// TIA Portal project "HydroPlantProject" (V15)

(* hardware
DEVICE "S71500/ET200MP station_1"  S7-1500 station
   slot 0: "Rail_0"  Rack  6ES7 590-1***0-0AA0
   slot 1: "PLC_1"  CPU 1511-1 PN  6ES7 511-1AK00-0AB0  V1.8
      slot 3: "CPU display_1"  6ES7591-1AA00-0AA0
DEVICE "PC-System_1"  SIMATIC PC station
   slot 0: "SIMATIC PC station"  Rail  SIMATIC PC-Station  V1.0
      slot 125: "Stationmanager"  Station_Manager  V6.0.4
   slot 1: "HMI_RT_1"  WinCC RT Professional  6AV2 105-0xxxx-xxxx  15.0.0.0
   slot 2: "IE general_1"  IE General  IE_CP  V8.2.0
*)

// ===== PLC "PLC_1"  CPU 1511-1 PN =====

VAR_GLOBAL   // PLC tag table "Default tag table"
   "Brake_Out" AT %M4.0 : Bool;
   "OilPumpVFDsp_Out" AT %MW6 : Int;
   "OilTemp_In" AT %MW12 : Int;
   "kW_In" AT %MW14 : Int;
   "RPM_In" AT %MW16 : Int;
   "Baffle_Out" AT %MW18 : Int;
   "OilPumpVFDen_Out" AT %M4.1 : Bool;
   "ProgLang" AT %MW0 : Int;
   "ONS1" AT %M2.0 : Bool;
   "PB_LAD" AT %M2.1 : Bool;
   "ONS" AT %M2.2 : Bool;
   "ONS2" AT %M2.3 : Bool;
   "ONS3" AT %M2.4 : Bool;
   "PB_FBD" AT %M2.5 : Bool;
   "PB_SCL" AT %M2.6 : Bool;
   "PB_STL" AT %M2.7 : Bool;
   "AlarmHorn_Out" AT %M3.0 : Bool;
   "StationInterlock_Out" AT %M3.1 : Bool;
   "OilPumpVFDpct" AT %MW8 : Int;
   "BafflePct" AT %MW10 : Int;
   "OilTemp" AT %MW20 : Int;
   "OilFlow" AT %MW22 : Int;
   "OilFlow_In" AT %MW24 : Int;
   "RPM" AT %MW26 : Int;
   "Current" AT %MW28 : Int;
   "Current_In" AT %MW30 : Int;
   "OilPumpVFDoff_Pb" AT %M3.2 : Bool;
   "OilPumpVFDhand_Pb" AT %M3.3 : Bool;
   "OilPumpVFDauto_Pb" AT %M3.4 : Bool;
   "BrakeOff_Pb" AT %M3.5 : Bool;
   "BrakeHand_Pb" AT %M3.6 : Bool;
   "BrakeAuto_Pb" AT %M3.7 : Bool;
   "BrakeHoa" AT %MW34 : Int;
   "AlarmHornOff_Pb" AT %M4.2 : Bool;
   "AlarmHornHand_Pb" AT %M4.3 : Bool;
   "AlarmHornAuto_Pb" AT %M4.4 : Bool;
   "AlarmHornHoa" AT %MW36 : Int;
   "StationIntOff_Pb" AT %M4.5 : Bool;
   "StationIntHand_Pb" AT %M4.6 : Bool;
   "StationIntAuto_Pb" AT %M4.7 : Bool;
   "StationIntHoa" AT %MW38 : Int;
   "OilPumpVFD_Ctrl" AT %M5.0 : Bool;
   "StationIntl_Ctrl" AT %M5.1 : Bool;
   "AlarmHorn_Ctrl" AT %M5.2 : Bool;
   "Brake_Ctrl" AT %M5.3 : Bool;
   "OilLowFlowDelay_Sp" AT %MW40 : Int;
   "AlarmReset" AT %M5.4 : Bool;
   "AlarmSilence" AT %M5.5 : Bool;
   "OilLowFlowAlarm" AT %M5.6 : Bool;
   "OilLowFlowNotify" AT %M5.7 : Bool;
   "OilLLflowSp" AT %MW42 : Int;
   "OvercurrentDelay_Sp" AT %MW44 : Int;
   "OvercurrentSp" AT %MW46 : Int;
   "OvercurrentAlarm" AT %M48.0 : Bool;
   "OvercurrentNotify" AT %M48.1 : Bool;
   "HighOilTempDelay_Sp" AT %MW50 : Int;
   "HighOilTempAlarm" AT %M48.2 : Bool;
   "HighOilTempNotify" AT %M48.3 : Bool;
   "HighOilTempSp" AT %MW52 : Int;
   "OverspeedDelay_Sp" AT %MW54 : Int;
   "OverspeedSp" AT %MW56 : Int;
   "OverspeedAlarm" AT %M48.4 : Bool;
   "OverspeedNotify" AT %M48.5 : Bool;
   "OilHighFlowDelay_Sp" AT %MW58 : Int;
   "OilHHflowSp" AT %MW60 : Int;
   "OilHighFlowAlarm" AT %M48.6 : Bool;
   "OilHighFlowNotify" AT %M48.7 : Bool;
   "BrakeFailureDelay_Sp" AT %MW62 : Int;
   "BrakeFailureAlarm" AT %M49.0 : Bool;
   "BrakeFailureNotify" AT %M49.1 : Bool;
   "EStop" AT %M49.2 : Bool;
   "EStopAlarm" AT %M49.3 : Bool;
   "EStopNotify" AT %M49.4 : Bool;
   "Tag_1" AT %T1 : Timer;
   "Tag_2" AT %T2 : Timer;
   "ONS2(1)" AT %M49.5 : Bool;
   "ONS2(2)" AT %M49.6 : Bool;
   "Baffle_En" AT %M49.7 : Bool;
   "Deleteme" AT %M64.0 : Bool;
   "deleteme1" AT %MD66 : Real;
   "WarmupMode" AT %M64.1 : Bool;
   "StabilizeMode" AT %M64.2 : Bool;
   "GenerationMode" AT %M64.3 : Bool;
   "CooldownMode" AT %M64.4 : Bool;
   "IdleMode" AT %M64.5 : Bool;
   "FaultMode" AT %M64.6 : Bool;
   "WarmupRPM" AT %MW70 : Int;
   "BafflePIDSp" AT %MW72 : Int;
   "BaffleHOA" AT %MW74 : Int;
   "Baffle_Ctrl" AT %M64.7 : Bool;
   "VFD_Sp" AT %MW76 : Int;
   "WarmupVFDpct" AT %MW78 : Int;
   "WarmupOilTemp" AT %MW80 : Int;
   "WarmupOilTempDelaySp" AT %MW82 : Int;
   "WarmupTrasition" AT %M65.0 : Bool;
   "BafflePIDin" AT %MW84 : Int;
   "StabilizekWSp" AT %MW86 : Int;
   "StabilizeDelaySp" AT %MW88 : Int;
   "StabilizeTrasition" AT %M65.1 : Bool;
   "SystemStart_Pb" AT %M65.2 : Bool;
   "StartSequenceBit" AT %M65.3 : Bool;
   "SystemStop_Pb" AT %M65.4 : Bool;
   "GenerationTransition" AT %M65.5 : Bool;
   "CooldownRPM" AT %MW90 : Int;
   "CooldownDelaySp" AT %MW92 : Int;
   "CooldownTrasition" AT %M65.6 : Bool;
   "CooldownRPMSp" AT %MW94 : Int;
   "CooldownOilTempSp" AT %MW96 : Int;
   "ONS4" AT %M65.7 : Bool;
   "SequenceRunning" AT %M98.0 : Bool;
   "ONS5" AT %M98.1 : Bool;
   "HOFoverrideVFDsp" AT %MW100 : Int;
   "ONS6" AT %M98.2 : Bool;
   "BaffleManual" AT %M98.3 : Bool;
   "BaffleAuto_Pb" AT %M98.4 : Bool;
   "BaffleHand_Pb" AT %M98.5 : Bool;
   "BaffleOff_Pb" AT %M98.6 : Bool;
   "ONS8" AT %M98.7 : Bool;
   "BaffleManualSp" AT %MD102 : Real;
   "ONS9" AT %M99.0 : Bool;
   "ONS10" AT %M99.1 : Bool;
   "ONS7" AT %M99.2 : Bool;
   "VFDHand_Pb" AT %M99.3 : Bool;
   "VFDOff_Pb" AT %M99.4 : Bool;
   "VFDAuto_Pb" AT %M99.5 : Bool;
   "ONS11" AT %M99.6 : Bool;
   "ONS12" AT %M99.7 : Bool;
   "ONS13" AT %M106.0 : Bool;
   "VFDHOA" AT %MW108 : Int;
   "VFDManualSp" AT %MD110 : Real;
   "ONS14" AT %M106.1 : Bool;
   "ONS15" AT %M106.2 : Bool;
   "VFDmanual" AT %M106.3 : Bool;
   "OilPumpVFDon" AT %M106.4 : Bool;
   "BafflePID_On" AT %M106.5 : Bool;
   "FullAutoBit" AT %M106.6 : Bool;
   "HM_Minutes" AT %MW32 : Int;
   "HM_Hours" AT %MW114 : Int;
   "HM_Days" AT %MW116 : Int;
   "ResetHourmeter_Pb" AT %M106.7 : Bool;
   "ModeInt" AT %MW118 : Int;
END_VAR

DATA_BLOCK "SimLogic_DB"   // DB1
{ S7_Optimized_Access := 'TRUE' }
VERSION : 0.1
// stored: InstanceOfName SimLogic
"SimLogic"
BEGIN
END_DATA_BLOCK

DATA_BLOCK "MODES_LAD_DB"   // DB2
{ S7_Optimized_Access := 'TRUE' }
VERSION : 0.1
// stored: InstanceOfName MODES_LAD
"MODES_LAD"
BEGIN
END_DATA_BLOCK

DATA_BLOCK "MODES_FBD_DB"   // DB4
{ S7_Optimized_Access := 'TRUE' }
VERSION : 0.1
// stored: InstanceOfName MODES_FBD
"MODES_FBD"
BEGIN
END_DATA_BLOCK

DATA_BLOCK "IO_LAD_DB"   // DB5
{ S7_Optimized_Access := 'TRUE' }
VERSION : 0.1
// stored: InstanceOfName IO_LAD
"IO_LAD"
BEGIN
END_DATA_BLOCK

DATA_BLOCK "IO_FBD_DB"   // DB6
{ S7_Optimized_Access := 'TRUE' }
VERSION : 0.1
// stored: InstanceOfName IO_FBD
"IO_FBD"
BEGIN
END_DATA_BLOCK

DATA_BLOCK "IO_SCL_DB"   // DB7
{ S7_Optimized_Access := 'TRUE' }
VERSION : 0.1
// stored: InstanceOfName IO_SCL
"IO_SCL"
BEGIN
END_DATA_BLOCK

DATA_BLOCK "IO_STL_DB"   // DB8
{ S7_Optimized_Access := 'TRUE' }
VERSION : 0.1
// stored: InstanceOfName IO_STL
"IO_STL"
BEGIN
END_DATA_BLOCK

DATA_BLOCK "ALARMS_LAD_DB"   // DB9
{ S7_Optimized_Access := 'TRUE' }
VERSION : 0.1
// stored: InstanceOfName ALARMS_LAD
"ALARMS_LAD"
BEGIN
END_DATA_BLOCK

DATA_BLOCK "HOA_LAD_DB"   // DB10
{ S7_Optimized_Access := 'TRUE' }
VERSION : 0.1
// stored: InstanceOfName HOA_LAD
"HOA_LAD"
BEGIN
END_DATA_BLOCK

DATA_BLOCK "HOA_FBD_DB"   // DB11
{ S7_Optimized_Access := 'TRUE' }
VERSION : 0.1
// stored: InstanceOfName HOA_FBD
"HOA_FBD"
BEGIN
END_DATA_BLOCK

DATA_BLOCK "HOA_SCL_DB"   // DB12
{ S7_Optimized_Access := 'TRUE' }
VERSION : 0.1
// stored: InstanceOfName HOA_SCL
"HOA_SCL"
BEGIN
END_DATA_BLOCK

DATA_BLOCK "HOA_STL_DB"   // DB13
{ S7_Optimized_Access := 'TRUE' }
VERSION : 0.1
// stored: InstanceOfName HOA_STL
"HOA_STL"
BEGIN
END_DATA_BLOCK

DATA_BLOCK "ALARMS_FBD_DB"   // DB14
{ S7_Optimized_Access := 'TRUE' }
VERSION : 0.1
// stored: InstanceOfName ALARMS_FBD
"ALARMS_FBD"
BEGIN
END_DATA_BLOCK

DATA_BLOCK "ALARMS_SCL_DB"   // DB15
{ S7_Optimized_Access := 'TRUE' }
VERSION : 0.1
// stored: InstanceOfName ALARMS_SCL
"ALARMS_SCL"
BEGIN
END_DATA_BLOCK

DATA_BLOCK "ALARMS_STL_DB"   // DB16
{ S7_Optimized_Access := 'TRUE' }
VERSION : 0.1
// stored: InstanceOfName ALARMS_STL
"ALARMS_STL"
BEGIN
END_DATA_BLOCK

DATA_BLOCK "MODES_SCL_DB"   // DB44
{ S7_Optimized_Access := 'TRUE' }
VERSION : 0.1
// stored: InstanceOfName MODES_SCL
"MODES_SCL"
BEGIN
END_DATA_BLOCK

DATA_BLOCK "MODES_STL_DB"   // DB45
{ S7_Optimized_Access := 'TRUE' }
VERSION : 0.1
// stored: InstanceOfName MODES_STL
"MODES_STL"
BEGIN
END_DATA_BLOCK

DATA_BLOCK "SEQUENCE_DB"   // DB58
{ S7_Optimized_Access := 'TRUE' }
VERSION : 0.1
// stored: InstanceOfName SEQUENCE
"SEQUENCE"
BEGIN
END_DATA_BLOCK

DATA_BLOCK "HOURMETER_LAD_DB"   // DB61
{ S7_Optimized_Access := 'TRUE' }
VERSION : 0.1
// stored: InstanceOfName HOURMETER_LAD
"HOURMETER_LAD"
BEGIN
END_DATA_BLOCK

DATA_BLOCK "HOURMETER_FBD_DB"   // DB62
{ S7_Optimized_Access := 'TRUE' }
VERSION : 0.1
// stored: InstanceOfName HOURMETER_FBD
"HOURMETER_FBD"
BEGIN
END_DATA_BLOCK

DATA_BLOCK "HOURMETER_SCL_DB"   // DB63
{ S7_Optimized_Access := 'TRUE' }
VERSION : 0.1
// stored: InstanceOfName HOURMETER_SCL
"HOURMETER_SCL"
BEGIN
END_DATA_BLOCK

DATA_BLOCK "HOURMETER_STL_DB"   // DB64
{ S7_Optimized_Access := 'TRUE' }
VERSION : 0.1
// stored: InstanceOfName HOURMETER_STL
"HOURMETER_STL"
BEGIN
END_DATA_BLOCK

// folder: System blocks/Program resources

DATA_BLOCK "IEC_Timer_0_DB_25"   // DB3
{ S7_Optimized_Access := 'TRUE' }
AUTHOR : Simatic
FAMILY : IEC
NAME : IEC_TMR
VERSION : 1.0
// stored: InstanceOfName IEC_TIMER
"IEC_TIMER"
BEGIN
END_DATA_BLOCK

DATA_BLOCK "IEC_Timer_0_DB"   // DB17
{ S7_Optimized_Access := 'TRUE' }
AUTHOR : Simatic
FAMILY : IEC
NAME : IEC_TMR
VERSION : 1.0
// stored: InstanceOfName IEC_TIMER
"IEC_TIMER"
BEGIN
END_DATA_BLOCK

DATA_BLOCK "IEC_Timer_0_DB_1"   // DB18
{ S7_Optimized_Access := 'TRUE' }
AUTHOR : Simatic
FAMILY : IEC
NAME : IEC_TMR
VERSION : 1.0
// stored: InstanceOfName IEC_TIMER
"IEC_TIMER"
BEGIN
END_DATA_BLOCK

DATA_BLOCK "IEC_Timer_0_DB_2"   // DB19
{ S7_Optimized_Access := 'TRUE' }
AUTHOR : Simatic
FAMILY : IEC
NAME : IEC_TMR
VERSION : 1.0
// stored: InstanceOfName IEC_TIMER
"IEC_TIMER"
BEGIN
END_DATA_BLOCK

DATA_BLOCK "IEC_Timer_0_DB_3"   // DB20
{ S7_Optimized_Access := 'TRUE' }
AUTHOR : Simatic
FAMILY : IEC
NAME : IEC_TMR
VERSION : 1.0
// stored: InstanceOfName IEC_TIMER
"IEC_TIMER"
BEGIN
END_DATA_BLOCK

DATA_BLOCK "IEC_Timer_0_DB_4"   // DB21
{ S7_Optimized_Access := 'TRUE' }
AUTHOR : Simatic
FAMILY : IEC
NAME : IEC_TMR
VERSION : 1.0
// stored: InstanceOfName IEC_TIMER
"IEC_TIMER"
BEGIN
END_DATA_BLOCK

DATA_BLOCK "IEC_Timer_0_DB_5"   // DB22
{ S7_Optimized_Access := 'TRUE' }
AUTHOR : Simatic
FAMILY : IEC
NAME : IEC_TMR
VERSION : 1.0
// stored: InstanceOfName IEC_TIMER
"IEC_TIMER"
BEGIN
END_DATA_BLOCK

DATA_BLOCK "IEC_Timer_0_DB_6"   // DB23
{ S7_Optimized_Access := 'TRUE' }
AUTHOR : Simatic
FAMILY : IEC
NAME : IEC_TMR
VERSION : 1.0
// stored: InstanceOfName IEC_TIMER
"IEC_TIMER"
BEGIN
END_DATA_BLOCK

DATA_BLOCK "IEC_Timer_0_DB_7"   // DB24
{ S7_Optimized_Access := 'TRUE' }
AUTHOR : Simatic
FAMILY : IEC
NAME : IEC_TMR
VERSION : 1.0
// stored: InstanceOfName IEC_TIMER
"IEC_TIMER"
BEGIN
END_DATA_BLOCK

DATA_BLOCK "IEC_Timer_0_DB_8"   // DB25
{ S7_Optimized_Access := 'TRUE' }
AUTHOR : Simatic
FAMILY : IEC
NAME : IEC_TMR
VERSION : 1.0
// stored: InstanceOfName IEC_TIMER
"IEC_TIMER"
BEGIN
END_DATA_BLOCK

DATA_BLOCK "IEC_Timer_0_DB_9"   // DB26
{ S7_Optimized_Access := 'TRUE' }
AUTHOR : Simatic
FAMILY : IEC
NAME : IEC_TMR
VERSION : 1.0
// stored: InstanceOfName IEC_TIMER
"IEC_TIMER"
BEGIN
END_DATA_BLOCK

DATA_BLOCK "IEC_Timer_0_DB_10"   // DB27
{ S7_Optimized_Access := 'TRUE' }
AUTHOR : Simatic
FAMILY : IEC
NAME : IEC_TMR
VERSION : 1.0
// stored: InstanceOfName IEC_TIMER
"IEC_TIMER"
BEGIN
END_DATA_BLOCK

DATA_BLOCK "IEC_Timer_0_DB_110"   // DB28
{ S7_Optimized_Access := 'TRUE' }
AUTHOR : Simatic
FAMILY : IEC
NAME : IEC_TMR
VERSION : 1.0
// stored: InstanceOfName IEC_TIMER
"IEC_TIMER"
BEGIN
END_DATA_BLOCK

DATA_BLOCK "IEC_Timer_0_DB_11"   // DB29
{ S7_Optimized_Access := 'TRUE' }
AUTHOR : Simatic
FAMILY : IEC
NAME : IEC_TMR
VERSION : 1.0
// stored: InstanceOfName IEC_TIMER
"IEC_TIMER"
BEGIN
END_DATA_BLOCK

DATA_BLOCK "IEC_Timer_0_DB_12"   // DB30
{ S7_Optimized_Access := 'TRUE' }
AUTHOR : Simatic
FAMILY : IEC
NAME : IEC_TMR
VERSION : 1.0
// stored: InstanceOfName IEC_TIMER
"IEC_TIMER"
BEGIN
END_DATA_BLOCK

DATA_BLOCK "IEC_Timer_0_DB_13"   // DB31
{ S7_Optimized_Access := 'TRUE' }
AUTHOR : Simatic
FAMILY : IEC
NAME : IEC_TMR
VERSION : 1.0
// stored: InstanceOfName IEC_TIMER
"IEC_TIMER"
BEGIN
END_DATA_BLOCK

DATA_BLOCK "IEC_Timer_0_DB_14"   // DB32
{ S7_Optimized_Access := 'TRUE' }
AUTHOR : Simatic
FAMILY : IEC
NAME : IEC_TMR
VERSION : 1.0
// stored: InstanceOfName IEC_TIMER
"IEC_TIMER"
BEGIN
END_DATA_BLOCK

DATA_BLOCK "IEC_Timer_0_DB_15"   // DB33
{ S7_Optimized_Access := 'TRUE' }
AUTHOR : Simatic
FAMILY : IEC
NAME : IEC_TMR
VERSION : 1.0
// stored: InstanceOfName IEC_TIMER
"IEC_TIMER"
BEGIN
END_DATA_BLOCK

DATA_BLOCK "IEC_Timer_0_DB_16"   // DB34
{ S7_Optimized_Access := 'TRUE' }
AUTHOR : Simatic
FAMILY : IEC
NAME : IEC_TMR
VERSION : 1.0
// stored: InstanceOfName IEC_TIMER
"IEC_TIMER"
BEGIN
END_DATA_BLOCK

DATA_BLOCK "IEC_Timer_0_DB_17"   // DB35
{ S7_Optimized_Access := 'TRUE' }
AUTHOR : Simatic
FAMILY : IEC
NAME : IEC_TMR
VERSION : 1.0
// stored: InstanceOfName IEC_TIMER
"IEC_TIMER"
BEGIN
END_DATA_BLOCK

DATA_BLOCK "IEC_Timer_0_DB_18"   // DB36
{ S7_Optimized_Access := 'TRUE' }
AUTHOR : Simatic
FAMILY : IEC
NAME : IEC_TMR
VERSION : 1.0
// stored: InstanceOfName IEC_TIMER
"IEC_TIMER"
BEGIN
END_DATA_BLOCK

DATA_BLOCK "IEC_Timer_0_DB_19"   // DB37
{ S7_Optimized_Access := 'TRUE' }
AUTHOR : Simatic
FAMILY : IEC
NAME : IEC_TMR
VERSION : 1.0
// stored: InstanceOfName IEC_TIMER
"IEC_TIMER"
BEGIN
END_DATA_BLOCK

DATA_BLOCK "IEC_Timer_0_DB_20"   // DB38
{ S7_Optimized_Access := 'TRUE' }
AUTHOR : Simatic
FAMILY : IEC
NAME : IEC_TMR
VERSION : 1.0
// stored: InstanceOfName IEC_TIMER
"IEC_TIMER"
BEGIN
END_DATA_BLOCK

DATA_BLOCK "IEC_Timer_0_DB_21"   // DB39
{ S7_Optimized_Access := 'TRUE' }
AUTHOR : Simatic
FAMILY : IEC
NAME : IEC_TMR
VERSION : 1.0
// stored: InstanceOfName IEC_TIMER
"IEC_TIMER"
BEGIN
END_DATA_BLOCK

DATA_BLOCK "IEC_Timer_0_DB_22"   // DB40
{ S7_Optimized_Access := 'TRUE' }
AUTHOR : Simatic
FAMILY : IEC
NAME : IEC_TMR
VERSION : 1.0
// stored: InstanceOfName IEC_TIMER
"IEC_TIMER"
BEGIN
END_DATA_BLOCK

DATA_BLOCK "IEC_Timer_0_DB_23"   // DB41
{ S7_Optimized_Access := 'TRUE' }
AUTHOR : Simatic
FAMILY : IEC
NAME : IEC_TMR
VERSION : 1.0
// stored: InstanceOfName IEC_TIMER
"IEC_TIMER"
BEGIN
END_DATA_BLOCK

DATA_BLOCK "IEC_Timer_1_DB"   // DB43
{ S7_Optimized_Access := 'TRUE' }
AUTHOR : Simatic
FAMILY : IEC
NAME : IEC_TMR
VERSION : 1.0
// stored: InstanceOfName IEC_TIMER
"IEC_TIMER"
BEGIN
END_DATA_BLOCK

DATA_BLOCK "IEC_Timer_0_DB_24"   // DB46
{ S7_Optimized_Access := 'TRUE' }
AUTHOR : Simatic
FAMILY : IEC
NAME : IEC_TMR
VERSION : 1.0
// stored: InstanceOfName IEC_TIMER
"IEC_TIMER"
BEGIN
END_DATA_BLOCK

DATA_BLOCK "IEC_Timer_0_DB_26"   // DB47
{ S7_Optimized_Access := 'TRUE' }
AUTHOR : Simatic
FAMILY : IEC
NAME : IEC_TMR
VERSION : 1.0
// stored: InstanceOfName IEC_TIMER
"IEC_TIMER"
BEGIN
END_DATA_BLOCK

DATA_BLOCK "IEC_Timer_0_DB_27"   // DB48
{ S7_Optimized_Access := 'TRUE' }
AUTHOR : Simatic
FAMILY : IEC
NAME : IEC_TMR
VERSION : 1.0
// stored: InstanceOfName IEC_TIMER
"IEC_TIMER"
BEGIN
END_DATA_BLOCK

DATA_BLOCK "IEC_Timer_0_DB_28"   // DB49
{ S7_Optimized_Access := 'TRUE' }
AUTHOR : Simatic
FAMILY : IEC
NAME : IEC_TMR
VERSION : 1.0
// stored: InstanceOfName IEC_TIMER
"IEC_TIMER"
BEGIN
END_DATA_BLOCK

DATA_BLOCK "IEC_Timer_0_DB_29"   // DB50
{ S7_Optimized_Access := 'TRUE' }
AUTHOR : Simatic
FAMILY : IEC
NAME : IEC_TMR
VERSION : 1.0
// stored: InstanceOfName IEC_TIMER
"IEC_TIMER"
BEGIN
END_DATA_BLOCK

DATA_BLOCK "IEC_Timer_0_DB_30"   // DB51
{ S7_Optimized_Access := 'TRUE' }
AUTHOR : Simatic
FAMILY : IEC
NAME : IEC_TMR
VERSION : 1.0
// stored: InstanceOfName IEC_TIMER
"IEC_TIMER"
BEGIN
END_DATA_BLOCK

DATA_BLOCK "IEC_Timer_0_DB_31"   // DB52
{ S7_Optimized_Access := 'TRUE' }
AUTHOR : Simatic
FAMILY : IEC
NAME : IEC_TMR
VERSION : 1.0
// stored: InstanceOfName IEC_TIMER
"IEC_TIMER"
BEGIN
END_DATA_BLOCK

DATA_BLOCK "IEC_Timer_0_DB_32"   // DB53
{ S7_Optimized_Access := 'TRUE' }
AUTHOR : Simatic
FAMILY : IEC
NAME : IEC_TMR
VERSION : 1.0
// stored: InstanceOfName IEC_TIMER
"IEC_TIMER"
BEGIN
END_DATA_BLOCK

DATA_BLOCK "IEC_Timer_0_DB_33"   // DB54
{ S7_Optimized_Access := 'TRUE' }
AUTHOR : Simatic
FAMILY : IEC
NAME : IEC_TMR
VERSION : 1.0
// stored: InstanceOfName IEC_TIMER
"IEC_TIMER"
BEGIN
END_DATA_BLOCK

DATA_BLOCK "IEC_Timer_0_DB_34"   // DB55
{ S7_Optimized_Access := 'TRUE' }
AUTHOR : Simatic
FAMILY : IEC
NAME : IEC_TMR
VERSION : 1.0
// stored: InstanceOfName IEC_TIMER
"IEC_TIMER"
BEGIN
END_DATA_BLOCK

DATA_BLOCK "IEC_Timer_0_DB_35"   // DB56
{ S7_Optimized_Access := 'TRUE' }
AUTHOR : Simatic
FAMILY : IEC
NAME : IEC_TMR
VERSION : 1.0
// stored: InstanceOfName IEC_TIMER
"IEC_TIMER"
BEGIN
END_DATA_BLOCK

DATA_BLOCK "IEC_Timer_0_DB_36"   // DB57
{ S7_Optimized_Access := 'TRUE' }
AUTHOR : Simatic
FAMILY : IEC
NAME : IEC_TMR
VERSION : 1.0
// stored: InstanceOfName IEC_TIMER
"IEC_TIMER"
BEGIN
END_DATA_BLOCK

DATA_BLOCK "IEC_Timer_0_DB_37"   // DB65
{ S7_Optimized_Access := 'TRUE' }
AUTHOR : Simatic
FAMILY : IEC
NAME : IEC_TMR
VERSION : 1.0
// stored: InstanceOfName IEC_TIMER
"IEC_TIMER"
BEGIN
END_DATA_BLOCK

DATA_BLOCK "IEC_Counter_0_DB"   // DB66
{ S7_Optimized_Access := 'TRUE' }
AUTHOR : Simatic
FAMILY : IEC
NAME : CNTR
VERSION : 1.0
// stored: InstanceOfName IEC_COUNTER
"IEC_COUNTER"
BEGIN
END_DATA_BLOCK

DATA_BLOCK "IEC_Counter_0_DB_1"   // DB67
{ S7_Optimized_Access := 'TRUE' }
AUTHOR : Simatic
FAMILY : IEC
NAME : CNTR
VERSION : 1.0
// stored: InstanceOfName IEC_COUNTER
"IEC_COUNTER"
BEGIN
END_DATA_BLOCK

DATA_BLOCK "IEC_Counter_0_DB_2"   // DB68
{ S7_Optimized_Access := 'TRUE' }
AUTHOR : Simatic
FAMILY : IEC
NAME : CNTR
VERSION : 1.0
// stored: InstanceOfName IEC_COUNTER
"IEC_COUNTER"
BEGIN
END_DATA_BLOCK

DATA_BLOCK "IEC_Timer_0_DB_38"   // DB69
{ S7_Optimized_Access := 'TRUE' }
AUTHOR : Simatic
FAMILY : IEC
NAME : IEC_TMR
VERSION : 1.0
// stored: InstanceOfName IEC_TIMER
"IEC_TIMER"
BEGIN
END_DATA_BLOCK

DATA_BLOCK "IEC_Timer_0_DB_39"   // DB70
{ S7_Optimized_Access := 'TRUE' }
AUTHOR : Simatic
FAMILY : IEC
NAME : IEC_TMR
VERSION : 1.0
// stored: InstanceOfName IEC_TIMER
"IEC_TIMER"
BEGIN
END_DATA_BLOCK

DATA_BLOCK "IEC_Timer_0_DB_40"   // DB71
{ S7_Optimized_Access := 'TRUE' }
AUTHOR : Simatic
FAMILY : IEC
NAME : IEC_TMR
VERSION : 1.0
// stored: InstanceOfName IEC_TIMER
"IEC_TIMER"
BEGIN
END_DATA_BLOCK

DATA_BLOCK "IEC_Counter_0_DB_3"   // DB72
{ S7_Optimized_Access := 'TRUE' }
AUTHOR : Simatic
FAMILY : IEC
NAME : CNTR
VERSION : 1.0
// stored: InstanceOfName IEC_COUNTER
"IEC_COUNTER"
BEGIN
END_DATA_BLOCK

DATA_BLOCK "IEC_Counter_0_DB_4"   // DB73
{ S7_Optimized_Access := 'TRUE' }
AUTHOR : Simatic
FAMILY : IEC
NAME : CNTR
VERSION : 1.0
// stored: InstanceOfName IEC_COUNTER
"IEC_COUNTER"
BEGIN
END_DATA_BLOCK

DATA_BLOCK "IEC_Counter_0_DB_5"   // DB74
{ S7_Optimized_Access := 'TRUE' }
AUTHOR : Simatic
FAMILY : IEC
NAME : CNTR
VERSION : 1.0
// stored: InstanceOfName IEC_COUNTER
"IEC_COUNTER"
BEGIN
END_DATA_BLOCK

DATA_BLOCK "IEC_Timer_0_DB_41"   // DB75
{ S7_Optimized_Access := 'TRUE' }
AUTHOR : Simatic
FAMILY : IEC
NAME : IEC_TMR
VERSION : 1.0
// stored: InstanceOfName IEC_TIMER
"IEC_TIMER"
BEGIN
END_DATA_BLOCK

DATA_BLOCK "IEC_Counter_0_DB_6"   // DB76
{ S7_Optimized_Access := 'TRUE' }
AUTHOR : Simatic
FAMILY : IEC
NAME : CNTR
VERSION : 1.0
// stored: InstanceOfName IEC_COUNTER
"IEC_COUNTER"
BEGIN
END_DATA_BLOCK

DATA_BLOCK "IEC_Counter_0_DB_7"   // DB77
{ S7_Optimized_Access := 'TRUE' }
AUTHOR : Simatic
FAMILY : IEC
NAME : CNTR
VERSION : 1.0
// stored: InstanceOfName IEC_COUNTER
"IEC_COUNTER"
BEGIN
END_DATA_BLOCK

DATA_BLOCK "IEC_Counter_0_DB_9"   // DB79
{ S7_Optimized_Access := 'TRUE' }
AUTHOR : Simatic
FAMILY : IEC
NAME : CNTR
VERSION : 1.0
// stored: InstanceOfName IEC_COUNTER
"IEC_COUNTER"
BEGIN
END_DATA_BLOCK

DATA_BLOCK "IEC_Timer_0_DB_42"   // DB80
{ S7_Optimized_Access := 'TRUE' }
AUTHOR : Simatic
FAMILY : IEC
NAME : IEC_TMR
VERSION : 1.0
// stored: InstanceOfName IEC_TIMER
"IEC_TIMER"
BEGIN
END_DATA_BLOCK

DATA_BLOCK "IEC_Timer_0_DB_43"   // DB81
{ S7_Optimized_Access := 'TRUE' }
AUTHOR : Simatic
FAMILY : IEC
NAME : IEC_TMR
VERSION : 1.0
// stored: InstanceOfName IEC_TIMER
"IEC_TIMER"
BEGIN
END_DATA_BLOCK

DATA_BLOCK "IEC_Counter_0_DB_10"   // DB82
{ S7_Optimized_Access := 'TRUE' }
AUTHOR : Simatic
FAMILY : IEC
NAME : CNTR
VERSION : 1.0
// stored: InstanceOfName IEC_COUNTER
"IEC_COUNTER"
BEGIN
END_DATA_BLOCK

DATA_BLOCK "IEC_Counter_0_DB_11"   // DB83
{ S7_Optimized_Access := 'TRUE' }
AUTHOR : Simatic
FAMILY : IEC
NAME : CNTR
VERSION : 1.0
// stored: InstanceOfName IEC_COUNTER
"IEC_COUNTER"
BEGIN
END_DATA_BLOCK

DATA_BLOCK "IEC_Counter_0_DB_12"   // DB84
{ S7_Optimized_Access := 'TRUE' }
AUTHOR : Simatic
FAMILY : IEC
NAME : CNTR
VERSION : 1.0
// stored: InstanceOfName IEC_COUNTER
"IEC_COUNTER"
BEGIN
END_DATA_BLOCK

DATA_BLOCK "IEC_Timer_0_DB_44"   // DB85
{ S7_Optimized_Access := 'TRUE' }
AUTHOR : Simatic
FAMILY : IEC
NAME : IEC_TMR
VERSION : 1.0
// stored: InstanceOfName IEC_TIMER
"IEC_TIMER"
BEGIN
END_DATA_BLOCK

// folder: (top level)

FUNCTION_BLOCK "SimLogic"   // FB1, LAD
{ S7_Optimized_Access := 'TRUE' }
VERSION : 0.1
   VAR
      "TO" : Bool;
      rpmv : Int;
      addrpmv : Bool;
      otsp : Int;
      ott : Int;
      TO1 : Bool;
      TO2 : Bool;
      be2 : Int;
      be3 : Int;
      be1 : Int;
      TO3 : Bool;
   END_VAR
   VAR_TEMP
      bf : Int;
      rpmvt : Int;
      bfr : Real;
   END_VAR
BEGIN

REGION Network 1
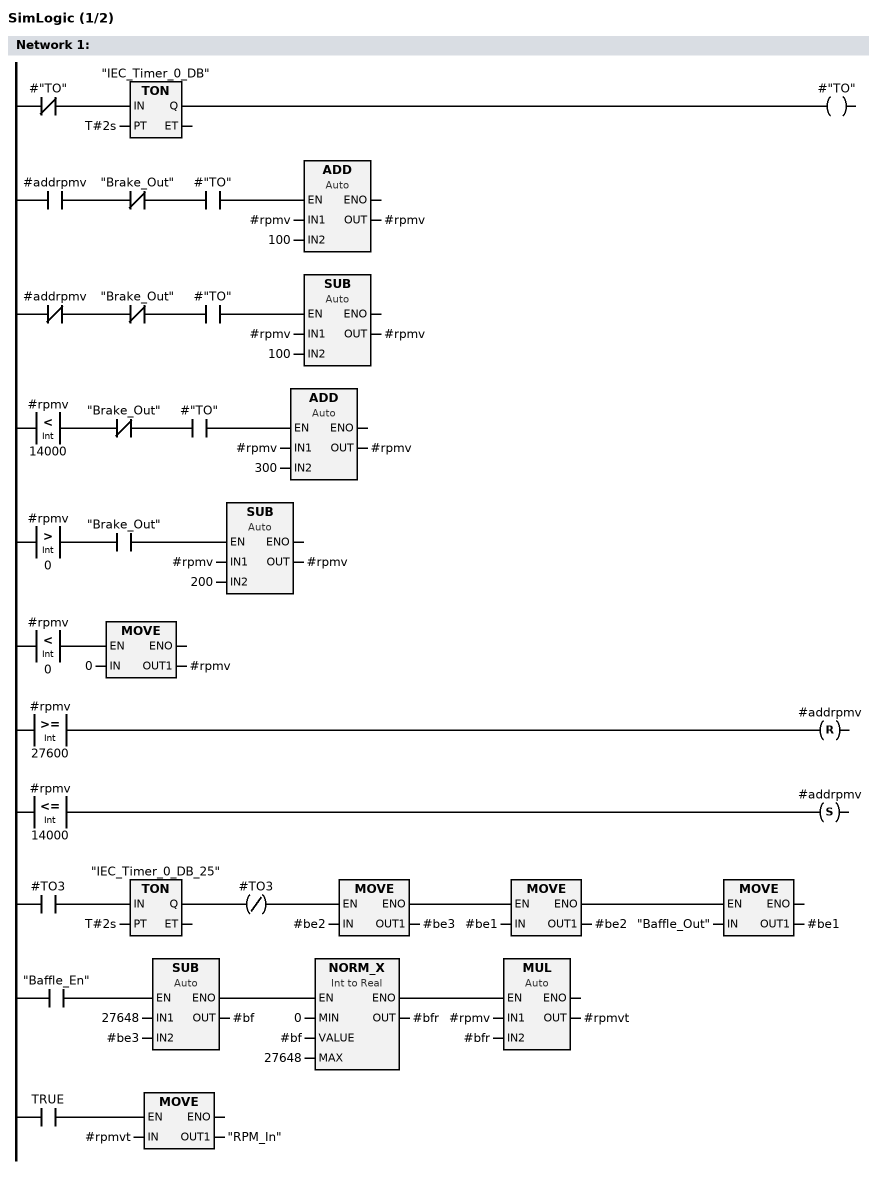
   "IEC_Timer_0_DB".TON(IN := NOT #"TO", PT := T#2s);
   #"TO" := "IEC_Timer_0_DB".Q;
   IF #addrpmv AND NOT "Brake_Out" AND #"TO" THEN #rpmv := #rpmv + 100; END_IF;
   IF NOT #addrpmv AND NOT "Brake_Out" AND #"TO" THEN #rpmv := #rpmv - 100; END_IF;
   IF (#rpmv < 14000) AND NOT "Brake_Out" AND #"TO" THEN #rpmv := #rpmv + 300; END_IF;
   IF (#rpmv > 0) AND "Brake_Out" THEN #rpmv := #rpmv - 200; END_IF;
   IF #rpmv < 0 THEN #rpmv := 0; END_IF;
   IF #rpmv >= 27600 THEN #addrpmv := FALSE; END_IF;
   IF #rpmv <= 14000 THEN #addrpmv := TRUE; END_IF;
   "IEC_Timer_0_DB_25".TON(IN := #TO3, PT := T#2s);
   #TO3 := NOT "IEC_Timer_0_DB_25".Q;
   IF "IEC_Timer_0_DB_25".Q THEN
       #be3 := #be2;
       #be2 := #be1;
       #be1 := "Baffle_Out";
   END_IF;
   IF "Baffle_En" THEN
       #bf := 27648 - #be3;
       #bfr := NORM_X(MIN := 0, VALUE := #bf, MAX := 27648);
       #rpmvt := #rpmv * #bfr;
   END_IF;
   IF TRUE THEN "RPM_In" := #rpmvt; END_IF;
END_REGION

REGION Network 2
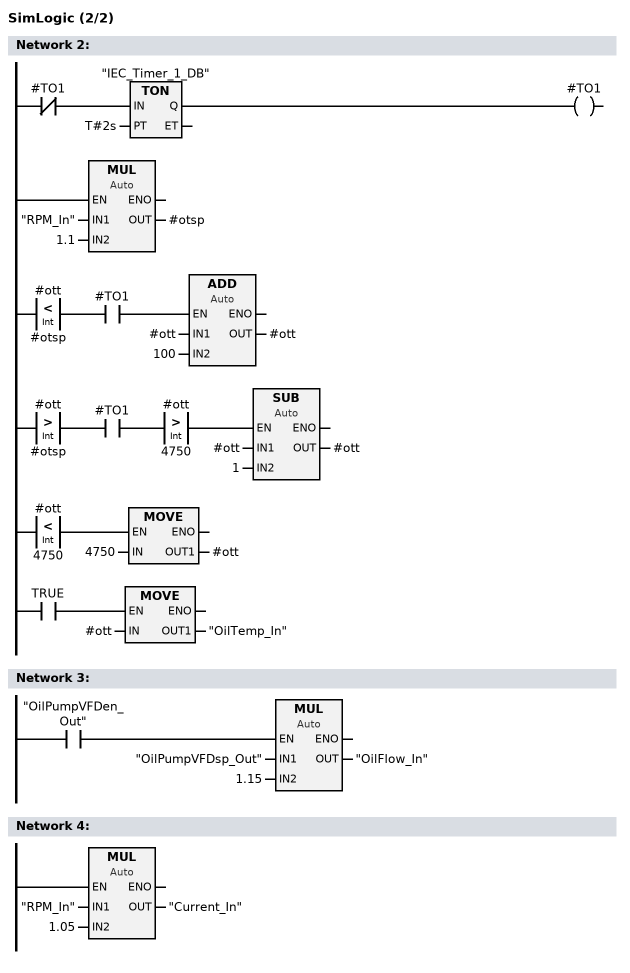
   "IEC_Timer_1_DB".TON(IN := NOT #TO1, PT := T#2s);
   #TO1 := "IEC_Timer_1_DB".Q;
   #otsp := "RPM_In" * 1.1;
   IF (#ott < #otsp) AND #TO1 THEN #ott := #ott + 100; END_IF;
   IF (#ott > #otsp) AND #TO1 AND (#ott > 4750) THEN #ott := #ott - 1; END_IF;
   IF #ott < 4750 THEN #ott := 4750; END_IF;
   IF TRUE THEN "OilTemp_In" := #ott; END_IF;
END_REGION

REGION Network 3
   RUNG wire#powerrail
      Contact( "OilPumpVFDen_Out" )
      Mul(in1 := "OilPumpVFDsp_Out", in2 := 1.15, out => "OilFlow_In")
   END_RUNG
   // the same network as SCL:
   IF "OilPumpVFDen_Out" THEN "OilFlow_In" := "OilPumpVFDsp_Out" * 1.15; END_IF;
END_REGION

REGION Network 4
   RUNG wire#powerrail
      Mul(in1 := "RPM_In", in2 := 1.05, out => "Current_In")
   END_RUNG
   // the same network as SCL:
   "Current_In" := "RPM_In" * 1.05;
END_REGION
END_FUNCTION_BLOCK

FUNCTION_BLOCK "IO_LAD"   // FB2, LAD
{ S7_Optimized_Access := 'TRUE' }
VERSION : 0.1
BEGIN

REGION Network 1
   // Digital Output
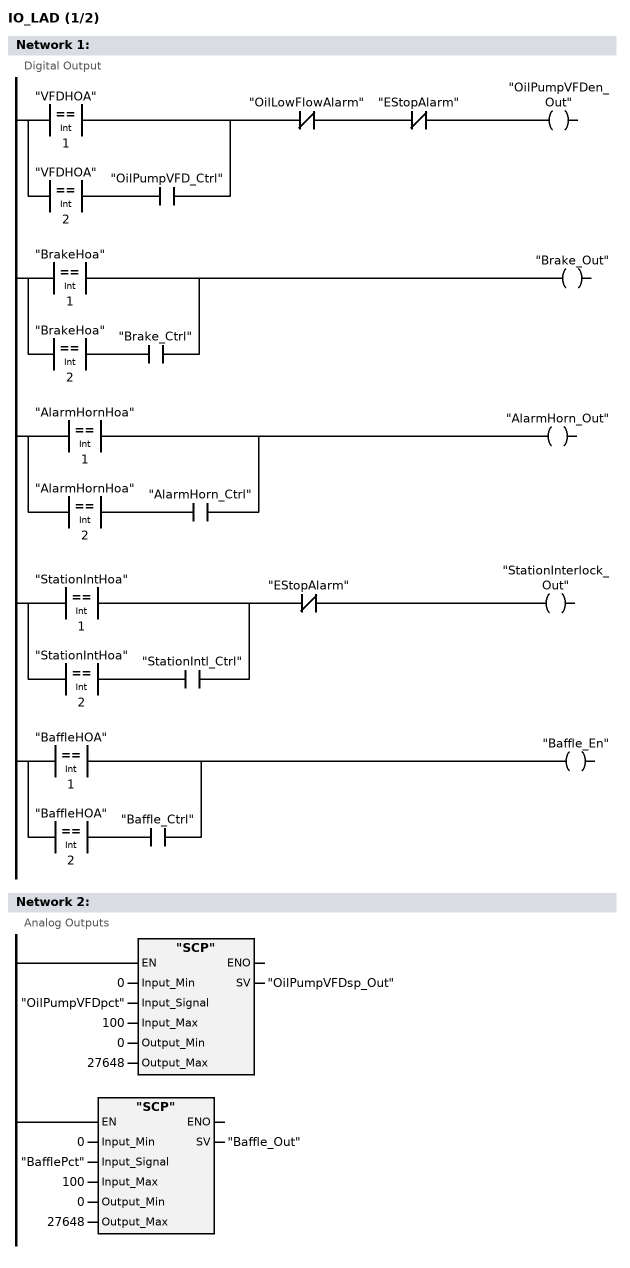
   RUNG wire#powerrail
      { S7_Templates := "SrcType := Int" } EQ_Contact(in1 := "VFDHOA", in2 := 1)
      wire#w1
      I_Contact( "OilLowFlowAlarm" )
      I_Contact( "EStopAlarm" )
      Coil( "OilPumpVFDen_Out" )
   END_RUNG
   RUNG wire#powerrail
      { S7_Templates := "SrcType := Int" } EQ_Contact(in1 := "VFDHOA", in2 := 2)
      Contact( "OilPumpVFD_Ctrl" )
   END_RUNG wire#w1
   RUNG wire#powerrail
      { S7_Templates := "SrcType := Int" } EQ_Contact(in1 := "BrakeHoa", in2 := 1)
      wire#w2
      Coil( "Brake_Out" )
   END_RUNG
   RUNG wire#powerrail
      { S7_Templates := "SrcType := Int" } EQ_Contact(in1 := "BrakeHoa", in2 := 2)
      Contact( "Brake_Ctrl" )
   END_RUNG wire#w2
   RUNG wire#powerrail
      { S7_Templates := "SrcType := Int" } EQ_Contact(in1 := "AlarmHornHoa", in2 := 1)
      wire#w3
      Coil( "AlarmHorn_Out" )
   END_RUNG
   RUNG wire#powerrail
      { S7_Templates := "SrcType := Int" } EQ_Contact(in1 := "AlarmHornHoa", in2 := 2)
      Contact( "AlarmHorn_Ctrl" )
   END_RUNG wire#w3
   RUNG wire#powerrail
      { S7_Templates := "SrcType := Int" } EQ_Contact(in1 := "StationIntHoa", in2 := 1)
      wire#w4
      I_Contact( "EStopAlarm" )
      Coil( "StationInterlock_Out" )
   END_RUNG
   RUNG wire#powerrail
      { S7_Templates := "SrcType := Int" } EQ_Contact(in1 := "StationIntHoa", in2 := 2)
      Contact( "StationIntl_Ctrl" )
   END_RUNG wire#w4
   RUNG wire#powerrail
      { S7_Templates := "SrcType := Int" } EQ_Contact(in1 := "BaffleHOA", in2 := 1)
      wire#w5
      Coil( "Baffle_En" )
   END_RUNG
   RUNG wire#powerrail
      { S7_Templates := "SrcType := Int" } EQ_Contact(in1 := "BaffleHOA", in2 := 2)
      Contact( "Baffle_Ctrl" )
   END_RUNG wire#w5
   // the same network as SCL:
   "OilPumpVFDen_Out" := (("VFDHOA" = 1) OR (("VFDHOA" = 2) AND "OilPumpVFD_Ctrl")) AND NOT "OilLowFlowAlarm" AND NOT "EStopAlarm";
   "Brake_Out" := ("BrakeHoa" = 1) OR (("BrakeHoa" = 2) AND "Brake_Ctrl");
   "AlarmHorn_Out" := ("AlarmHornHoa" = 1) OR (("AlarmHornHoa" = 2) AND "AlarmHorn_Ctrl");
   "StationInterlock_Out" := (("StationIntHoa" = 1) OR (("StationIntHoa" = 2) AND "StationIntl_Ctrl")) AND NOT "EStopAlarm";
   "Baffle_En" := ("BaffleHOA" = 1) OR (("BaffleHOA" = 2) AND "Baffle_Ctrl");
END_REGION

REGION Network 2
   // Analog Outputs
   RUNG wire#powerrail
      "SCP"(Input_Min := 0, Input_Signal := "OilPumpVFDpct", Input_Max := 100, Output_Min := 0, Output_Max := 27648, SV => "OilPumpVFDsp_Out")
   END_RUNG
   RUNG wire#powerrail
      "SCP"(Input_Min := 0, Input_Signal := "BafflePct", Input_Max := 100, Output_Min := 0, Output_Max := 27648, SV => "Baffle_Out")
   END_RUNG
   // the same network as SCL:
   "SCP"(Input_Min := 0,
         Input_Signal := "OilPumpVFDpct",
         Input_Max := 100,
         Output_Min := 0,
         Output_Max := 27648,
         SV => "OilPumpVFDsp_Out");
   "SCP"(Input_Min := 0,
         Input_Signal := "BafflePct",
         Input_Max := 100,
         Output_Min := 0,
         Output_Max := 27648,
         SV => "Baffle_Out");
END_REGION

REGION Network 3
   // Analog Inputs
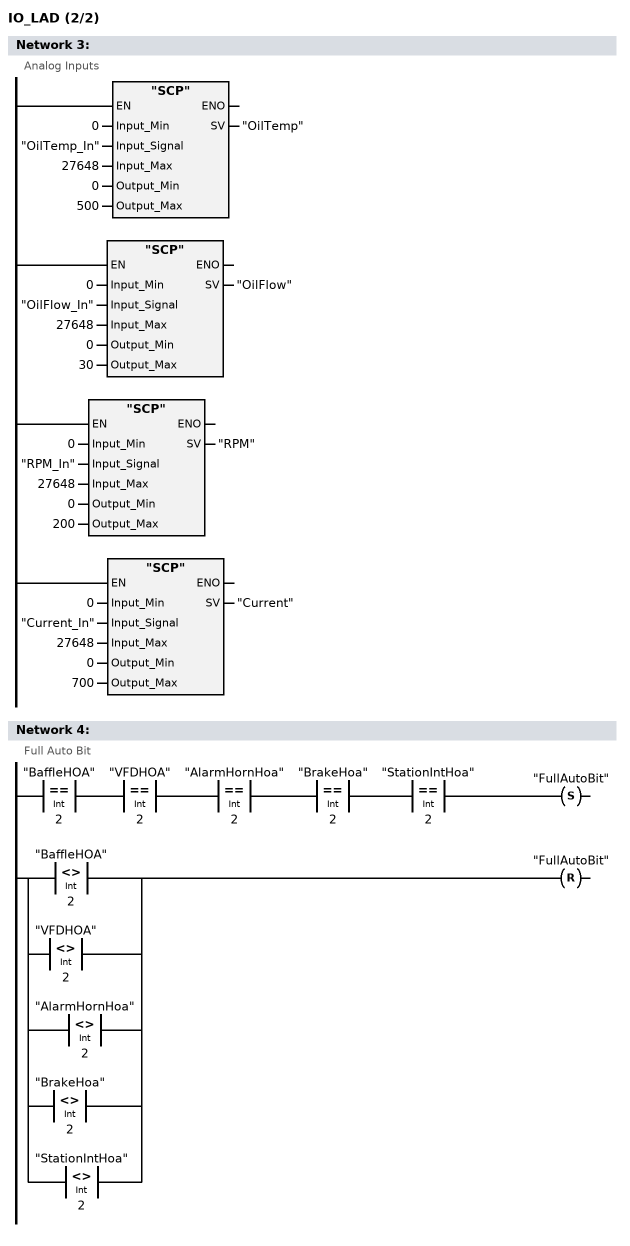
   RUNG wire#powerrail
      "SCP"(Input_Min := 0, Input_Signal := "OilTemp_In", Input_Max := 27648, Output_Min := 0, Output_Max := 500, SV => "OilTemp")
   END_RUNG
   RUNG wire#powerrail
      "SCP"(Input_Min := 0, Input_Signal := "OilFlow_In", Input_Max := 27648, Output_Min := 0, Output_Max := 30, SV => "OilFlow")
   END_RUNG
   RUNG wire#powerrail
      "SCP"(Input_Min := 0, Input_Signal := "RPM_In", Input_Max := 27648, Output_Min := 0, Output_Max := 200, SV => "RPM")
   END_RUNG
   RUNG wire#powerrail
      "SCP"(Input_Min := 0, Input_Signal := "Current_In", Input_Max := 27648, Output_Min := 0, Output_Max := 700, SV => "Current")
   END_RUNG
   // the same network as SCL:
   "SCP"(Input_Min := 0,
         Input_Signal := "OilTemp_In",
         Input_Max := 27648,
         Output_Min := 0,
         Output_Max := 500,
         SV => "OilTemp");
   "SCP"(Input_Min := 0,
         Input_Signal := "OilFlow_In",
         Input_Max := 27648,
         Output_Min := 0,
         Output_Max := 30,
         SV => "OilFlow");
   "SCP"(Input_Min := 0,
         Input_Signal := "RPM_In",
         Input_Max := 27648,
         Output_Min := 0,
         Output_Max := 200,
         SV => "RPM");
   "SCP"(Input_Min := 0,
         Input_Signal := "Current_In",
         Input_Max := 27648,
         Output_Min := 0,
         Output_Max := 700,
         SV => "Current");
END_REGION

REGION Network 4
   // Full Auto Bit
   RUNG wire#powerrail
      { S7_Templates := "SrcType := Int" } EQ_Contact(in1 := "BaffleHOA", in2 := 2)
      { S7_Templates := "SrcType := Int" } EQ_Contact(in1 := "VFDHOA", in2 := 2)
      { S7_Templates := "SrcType := Int" } EQ_Contact(in1 := "AlarmHornHoa", in2 := 2)
      { S7_Templates := "SrcType := Int" } EQ_Contact(in1 := "BrakeHoa", in2 := 2)
      { S7_Templates := "SrcType := Int" } EQ_Contact(in1 := "StationIntHoa", in2 := 2)
      S_Coil( "FullAutoBit" )
   END_RUNG
   RUNG wire#powerrail
      { S7_Templates := "SrcType := Int" } NE_Contact(in1 := "BaffleHOA", in2 := 2)
      wire#w1
      R_Coil( "FullAutoBit" )
   END_RUNG
   RUNG wire#powerrail
      { S7_Templates := "SrcType := Int" } NE_Contact(in1 := "VFDHOA", in2 := 2)
   END_RUNG wire#w1
   RUNG wire#powerrail
      { S7_Templates := "SrcType := Int" } NE_Contact(in1 := "AlarmHornHoa", in2 := 2)
   END_RUNG wire#w1
   RUNG wire#powerrail
      { S7_Templates := "SrcType := Int" } NE_Contact(in1 := "BrakeHoa", in2 := 2)
   END_RUNG wire#w1
   RUNG wire#powerrail
      { S7_Templates := "SrcType := Int" } NE_Contact(in1 := "StationIntHoa", in2 := 2)
   END_RUNG wire#w1
   // the same network as SCL:
   IF ("BaffleHOA" = 2) AND ("VFDHOA" = 2) AND ("AlarmHornHoa" = 2) AND ("BrakeHoa" = 2) AND ("StationIntHoa" = 2) THEN
       "FullAutoBit" := TRUE;
   END_IF;
   IF ("BaffleHOA" <> 2) OR ("VFDHOA" <> 2) OR ("AlarmHornHoa" <> 2) OR ("BrakeHoa" <> 2) OR ("StationIntHoa" <> 2) THEN
       "FullAutoBit" := FALSE;
   END_IF;
END_REGION
END_FUNCTION_BLOCK

FUNCTION_BLOCK "IO_FBD"   // FB3, FBD
{ S7_Optimized_Access := 'TRUE' }
VERSION : 0.1
   VAR_TEMP
      tv : Real;
   END_VAR
BEGIN

REGION Network 1
   // Digital Outputs
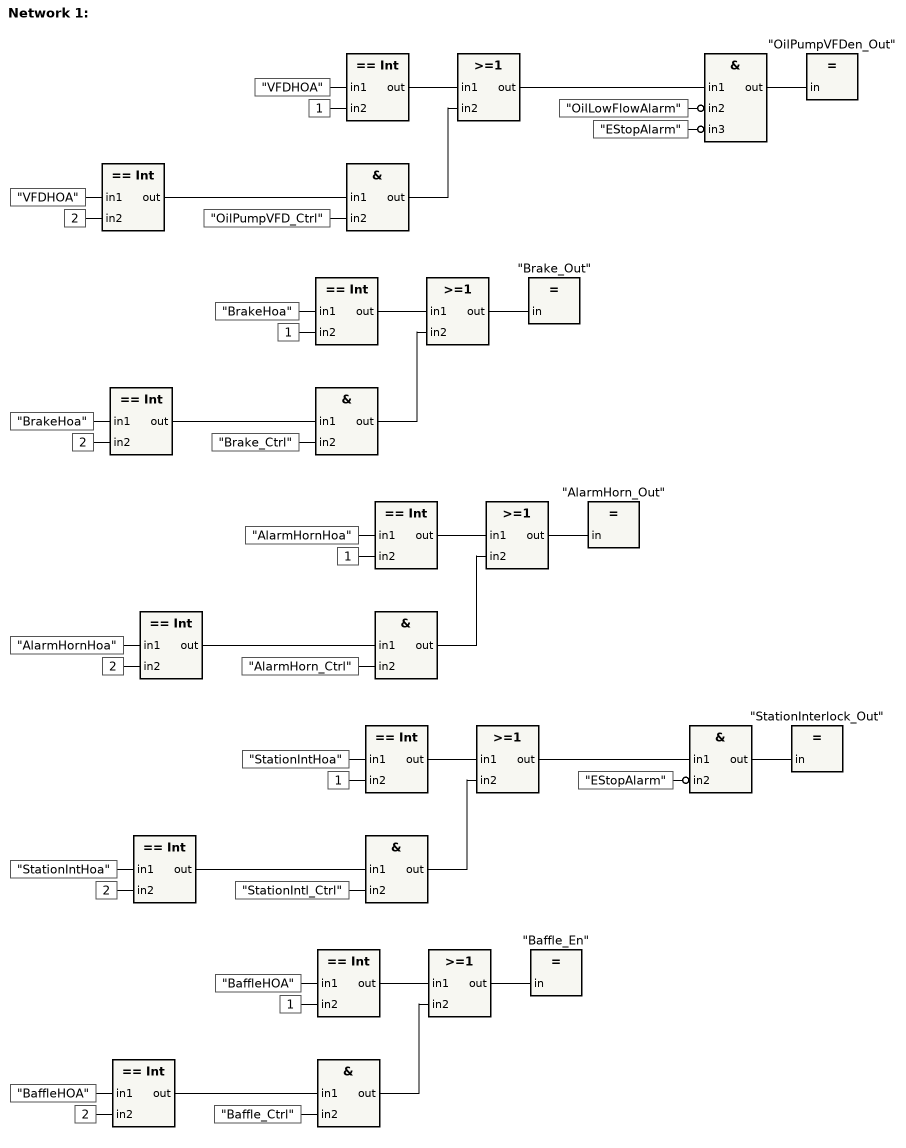
   "OilPumpVFDen_Out" := (("VFDHOA" = 1) OR (("VFDHOA" = 2) AND "OilPumpVFD_Ctrl")) AND NOT "OilLowFlowAlarm" AND NOT "EStopAlarm";
   "Brake_Out" := ("BrakeHoa" = 1) OR (("BrakeHoa" = 2) AND "Brake_Ctrl");
   "AlarmHorn_Out" := ("AlarmHornHoa" = 1) OR (("AlarmHornHoa" = 2) AND "AlarmHorn_Ctrl");
   "StationInterlock_Out" := (("StationIntHoa" = 1) OR (("StationIntHoa" = 2) AND "StationIntl_Ctrl")) AND NOT "EStopAlarm";
   "Baffle_En" := ("BaffleHOA" = 1) OR (("BaffleHOA" = 2) AND "Baffle_Ctrl");
END_REGION

REGION Network 2
   // Analog Outputs
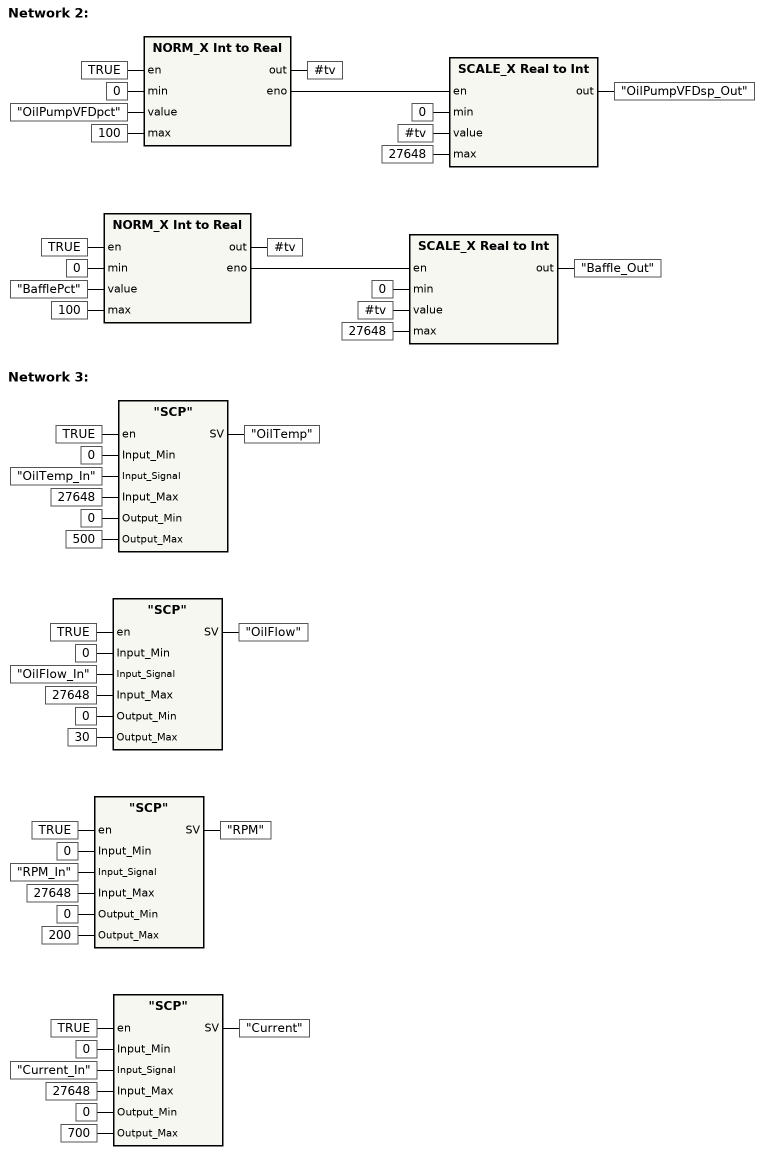
   IF TRUE THEN
       #tv := NORM_X(MIN := 0, VALUE := "OilPumpVFDpct", MAX := 100);
       "OilPumpVFDsp_Out" := SCALE_X(MIN := 0, VALUE := #tv, MAX := 27648);
       #tv := NORM_X(MIN := 0, VALUE := "BafflePct", MAX := 100);
       "Baffle_Out" := SCALE_X(MIN := 0, VALUE := #tv, MAX := 27648);
   END_IF;
END_REGION

REGION Network 3
   // Analog Inputs
   IF TRUE THEN
       "SCP"(Input_Min := 0,
             Input_Signal := "OilTemp_In",
             Input_Max := 27648,
             Output_Min := 0,
             Output_Max := 500,
             SV => "OilTemp");
       "SCP"(Input_Min := 0,
             Input_Signal := "OilFlow_In",
             Input_Max := 27648,
             Output_Min := 0,
             Output_Max := 30,
             SV => "OilFlow");
       "SCP"(Input_Min := 0,
             Input_Signal := "RPM_In",
             Input_Max := 27648,
             Output_Min := 0,
             Output_Max := 200,
             SV => "RPM");
       "SCP"(Input_Min := 0,
             Input_Signal := "Current_In",
             Input_Max := 27648,
             Output_Min := 0,
             Output_Max := 700,
             SV => "Current");
   END_IF;
END_REGION

REGION Network 4
   // Full Auto Bit
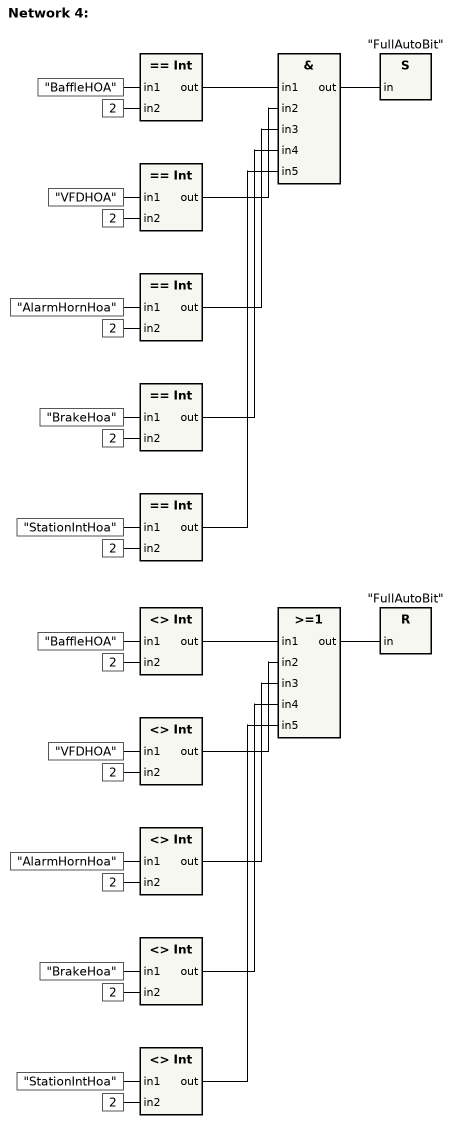
   IF ("BaffleHOA" = 2) AND ("VFDHOA" = 2) AND ("AlarmHornHoa" = 2) AND ("BrakeHoa" = 2) AND ("StationIntHoa" = 2) THEN
       "FullAutoBit" := TRUE;
   END_IF;
   IF ("BaffleHOA" <> 2) OR ("VFDHOA" <> 2) OR ("AlarmHornHoa" <> 2) OR ("BrakeHoa" <> 2) OR ("StationIntHoa" <> 2) THEN
       "FullAutoBit" := FALSE;
   END_IF;
END_REGION
END_FUNCTION_BLOCK

FUNCTION_BLOCK "IO_SCL"   // FB4, SCL
{ S7_Optimized_Access := 'TRUE' }
VERSION : 0.1
BEGIN
   //Digital Outputs
   IF "EStopAlarm" OR "OilLowFlowAlarm" OR "VFDHOA" = 0 OR ("VFDHOA" = 2 AND NOT "OilPumpVFD_Ctrl") THEN
       "OilPumpVFDen_Out" := 0;
   END_IF;

   IF ("VFDHOA" = 1 OR ("VFDHOA" = 2 AND "OilPumpVFD_Ctrl")) AND NOT "OilLowFlowAlarm" AND NOT "EStopAlarm" THEN
       "OilPumpVFDen_Out" := 1;
   END_IF;

   IF "BrakeHoa" = 0 OR ("BrakeHoa" = 2 AND NOT "Brake_Ctrl") THEN
       "Brake_Out" := 0;
   END_IF;

   IF "BrakeHoa" = 1 OR ("BrakeHoa" = 2 AND "Brake_Ctrl") THEN
       "Brake_Out" := 1;
   END_IF;

   IF "AlarmHornHoa" = 0 OR ("AlarmHornHoa" = 2 AND NOT "AlarmHorn_Ctrl") THEN
       "AlarmHorn_Out" := 0;
   END_IF;

   IF "AlarmHornHoa" = 1 OR ("AlarmHornHoa" = 2 AND "AlarmHorn_Ctrl") THEN
       "AlarmHorn_Out" := 1;
   END_IF;

   IF "StationIntHoa" = 0 OR ("StationIntHoa" = 2 AND NOT "StationIntl_Ctrl") THEN
       "StationInterlock_Out" := 0;
   END_IF;

   IF "StationIntHoa" = 1 OR ("StationIntHoa" = 2 AND "StationIntl_Ctrl") THEN
       "StationInterlock_Out" := 1;
   END_IF;

   IF "BaffleHOA" = 0 OR ("BaffleHOA" = 2 AND NOT "Baffle_Ctrl") THEN
       "Baffle_En" := 0;
   END_IF;

   IF "BaffleHOA" = 1 OR ("BaffleHOA" = 2 AND "Baffle_Ctrl") THEN
       "Baffle_En" := 1;
   END_IF;





   //Analog Outputs
   "SCP"(Input_Min:=0,
         Input_Signal:="OilPumpVFDpct",
         Input_Max:=100,
         Output_Min:=0,
         Output_Max:=27648,
         SV=>"OilPumpVFDsp_Out");

   "SCP"(Input_Min := 0,
         Input_Signal := "BafflePct",
         Input_Max := 100,
         Output_Min := 0,
         Output_Max := 27648,
         SV => "Baffle_Out");


   //Analog Inputs
   "SCP"(Input_Min:=0,
         Input_Signal:="OilTemp_In",
         Input_Max:=27648,
         Output_Min:=0,
         Output_Max:=500,
         SV=>"OilTemp");

   "SCP"(Input_Min := 0,
         Input_Signal := "OilFlow_In",
         Input_Max := 27648,
         Output_Min := 0,
         Output_Max := 30,
         SV => "OilFlow");

   "SCP"(Input_Min := 0,
         Input_Signal := "RPM_In",
         Input_Max := 27648,
   Output_Min := 0,
   Output_Max := 200,
   SV => "RPM");

   "SCP"(Input_Min := 0,
         Input_Signal := "Current_In",
         Input_Max := 27648,
         Output_Min := 0,
         Output_Max := 700,
         SV => "Current");


   //Full Auto Bit
   IF "BaffleHOA" = 2 AND "AlarmHornHoa" = 2 AND "VFDHOA" = 2 AND "StationIntHoa" = 2 AND "BrakeHoa" = 2 THEN
       "FullAutoBit" := 1;
   ELSE
       "FullAutoBit" := 0;
   END_IF;
END_FUNCTION_BLOCK

FUNCTION_BLOCK "IO_STL"   // FB5, STL
{ S7_Optimized_Access := 'TRUE' }
VERSION : 0.1
BEGIN

REGION Network 1
   //Digital Outputs
         A     "OilLowFlowAlarm";
         JC    ResetOilPumpVFD;
         CLR;
         A     "EStopAlarm";
         JC    ResetOilPumpVFD;
         L     "VFDHOA";
         L     0;
         ==I;
         JC    ResetOilPumpVFD;
         CLR;
         L     "VFDHOA";
         L     1;
         ==I;
         JC    SetOilPumpVFD;
         CLR;
         L     "VFDHOA";
         L     2;
         ==I;
         JC    AutoOilPumpVFD;

   AutoOilPumpVFD:A     "OilPumpVFD_Ctrl";
         JC    SetOilPumpVFD;
         JU    ResetOilPumpVFD;

   SetOilPumpVFD:AN    "OilLowFlowAlarm";
         AN    "EStop";
         S     "OilPumpVFDen_Out";
         JU    Brake;

   ResetOilPumpVFD:R     "OilPumpVFDen_Out";
         JU    Brake;

   Brake:L     "BrakeHoa";
         L     0;
         ==I;
         JC    ResetBrake;
         CLR;
         L     "BrakeHoa";
         L     1;
         ==I;
         JC    SetBrake;
         CLR;
         L     "BrakeHoa";
         L     2;
         ==I;
         JC    AutoBrake;

   AutoBrake:A     "Brake_Ctrl";
         JC    SetBrake;
         JU    ResetBrake;

   SetBrake:S     "Brake_Out";
         JU    AlarmHorn;

   ResetBrake:R     "Brake_Out";
         JU    AlarmHorn;

   AlarmHorn:L     "AlarmHornHoa";
         L     0;
         ==I;
         JC    ResetAlarmHorn;
         CLR;
         L     "AlarmHornHoa";
         L     1;
         ==I;
         JC    SetAlarmHorn;
         CLR;
         L     "AlarmHornHoa";
         L     2;
         ==I;
         JC    AutoAlarmHorn;

   AutoAlarmHorn:A     "AlarmHorn_Ctrl";
         JC    SetAlarmHorn;
         JU    ResetAlarmHorn;

   SetAlarmHorn:S     "AlarmHorn_Out";
         JU    StationInterlock;

   ResetAlarmHorn:R     "AlarmHorn_Out";
         JU    StationInterlock;

   StationInterlock:A     "EStopAlarm";
         JC    ResetStationInterlock;
         L     "StationIntHoa";
         L     0;
         ==I;
         JC    ResetStationInterlock;
         CLR;
         L     "StationIntHoa";
         L     1;
         ==I;
         JC    SetStationInterlock;
         CLR;
         L     "StationIntHoa";
         L     2;
         ==I;
         JC    AutoStationInterlock;

   AutoStationInterlock:A     "StationIntl_Ctrl";
         JC    SetStationInterlock;
         JU    ResetStationInterlock;

   SetStationInterlock:AN    "EStopAlarm";
         S     "StationInterlock_Out";
         JU    Baffle;

   ResetStationInterlock:R     "StationInterlock_Out";
         JU    Baffle;

   Baffle:L     "BaffleHOA";
         L     0;
         ==I;
         JC    ResetBaffle;
         CLR;
         L     "BaffleHOA";
         L     1;
         ==I;
         JC    SetBaffle;
         CLR;
         L     "BaffleHOA";
         L     2;
         ==I;
         JC    AutoBaffle;

   AutoBaffle:A     "Baffle_Ctrl";
         JC    SetBaffle;
         JU    ResetBaffle;

   SetBaffle:S     "Baffle_En";
         JU    AnalogOutputs;

   ResetBaffle:R     "Baffle_En";
         JU    AnalogOutputs;



   //Analog Outputs
   AnalogOutputs:CALL  "SCP"
         ( Input_Min    := 0,
           Input_Signal := "OilPumpVFDpct",
           Input_Max    := 100,
           Output_Min   := 0,
           Output_Max   := 27648,
           SV           := "OilPumpVFDsp_Out"
         );
         JU    AnalogInputs;

         CALL  "SCP"
         ( Input_Min    := 0,
           Input_Signal := "BafflePct",
           Input_Max    := 100,
           Output_Min   := 0,
           Output_Max   := 27648,
           SV           := "Baffle_Out"
         );


   //Analog Inputs
   AnalogInputs:CALL  "SCP"
         ( Input_Min    := 0,
           Input_Signal := "OilTemp_In",
           Input_Max    := 27648,
           Output_Min   := 0,
           Output_Max   := 500,
           SV           := "OilTemp"
         );

         CALL  "SCP"
         ( Input_Min    := 0,
           Input_Signal := "OilFlow_In",
           Input_Max    := 27648,
           Output_Min   := 0,
           Output_Max   := 30,
           SV           := "OilFlow"
         );

         CALL  "SCP"
         ( Input_Min    := 0,
           Input_Signal := "RPM_In",
           Input_Max    := 27648,
           Output_Min   := 0,
           Output_Max   := 200,
           SV           := "RPM"
         );

         CALL  "SCP"
         ( Input_Min    := 0,
           Input_Signal := "Current_In",
           Input_Max    := 27648,
           Output_Min   := 0,
           Output_Max   := 700,
           SV           := "Current"
         );

   //Full Auto Bit
         CLR;
         L     "BaffleHOA";
         L     2;
         ==I;
         NOT;
         JC    ResetFullAuto;
         CLR;
         L     "VFDHOA";
         L     2;
         ==I;
         NOT;
         JC    ResetFullAuto;
         CLR;
         L     "AlarmHornHoa";
         L     2;
         ==I;
         NOT;
         JC    ResetFullAuto;
         CLR;
         L     "BrakeHoa";
         L     2;
         ==I;
         NOT;
         JC    ResetFullAuto;
         CLR;
         L     "StationIntHoa";
         L     2;
         ==I;
         NOT;
         JC    ResetFullAuto;
         CLR;
         SET;
         S     "FullAutoBit";
         JU    EndOfLine;

   ResetFullAuto:SET;
         NOT;
         R     "FullAutoBit";
         JU    EndOfLine;

   EndOfLine:BE;
END_REGION
END_FUNCTION_BLOCK

FUNCTION_BLOCK "ALARMS_LAD"   // FB6, LAD
{ S7_Optimized_Access := 'TRUE' }
VERSION : 0.1
   VAR
      OS1 : Bool;
      OS2 : Bool;
      OS3 : Bool;
      OS4 : Bool;
      OS5 : Bool;
      OS6 : Bool;
      OS7 : Bool;
      OS8 : Bool;
   END_VAR
   VAR_TEMP
      tv : Time;
      Tsp : Int;
      OLFAT : Bool;
      OLFD : Int;
      tv1 : Time;
      OCD : Int;
      tv2 : Time;
      OCAT : Bool;
      HOTD : Int;
      tv3 : Time;
      HOTAT : Bool;
      OSD : Int;
      tv4 : Time;
      OSAT : Bool;
      OHFD : Int;
      tv5 : Time;
      OHFAT : Bool;
      BFD : Int;
      tv6 : Time;
      BFAT : Bool;
      ESAT : Bool;
      AlarmHornTrigger : Bool;
   END_VAR
   VAR_TEMP   // added for the SCL form of the ladder/FBD networks
      _w1 : Bool;
   END_VAR
BEGIN

REGION Network 1
   // Oil Low Flow Alarm
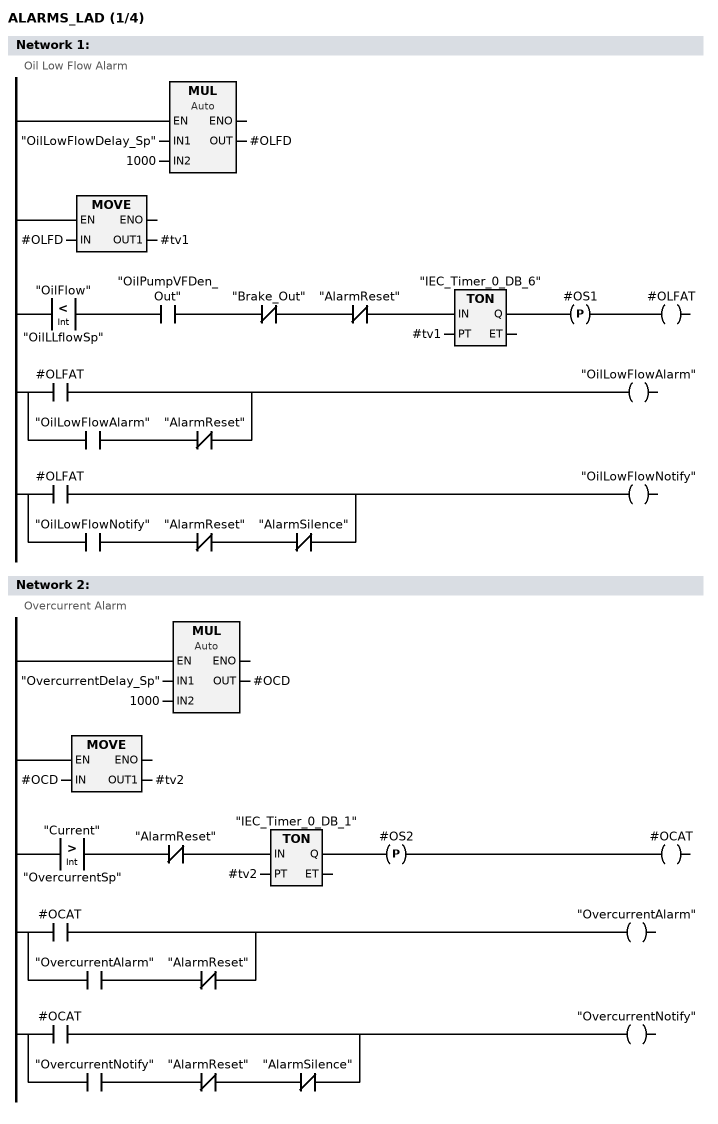
   #OLFD := "OilLowFlowDelay_Sp" * 1000;
   #tv1 := #OLFD;
   "IEC_Timer_0_DB_6".TON(IN := ("OilFlow" < "OilLLflowSp") AND "OilPumpVFDen_Out" AND NOT "Brake_Out" AND NOT "AlarmReset",
                          PT := #tv1);
   #_w1 := "IEC_Timer_0_DB_6".Q AND NOT #OS1;   // rising edge
   #OS1 := "IEC_Timer_0_DB_6".Q;
   #OLFAT := #_w1;
   "OilLowFlowAlarm" := #OLFAT OR ("OilLowFlowAlarm" AND NOT "AlarmReset");
   "OilLowFlowNotify" := #OLFAT OR ("OilLowFlowNotify" AND NOT "AlarmReset" AND NOT "AlarmSilence");
END_REGION

REGION Network 2
   // Overcurrent Alarm
   #OCD := "OvercurrentDelay_Sp" * 1000;
   #tv2 := #OCD;
   "IEC_Timer_0_DB_1".TON(IN := ("Current" > "OvercurrentSp") AND NOT "AlarmReset", PT := #tv2);
   #_w1 := "IEC_Timer_0_DB_1".Q AND NOT #OS2;   // rising edge
   #OS2 := "IEC_Timer_0_DB_1".Q;
   #OCAT := #_w1;
   "OvercurrentAlarm" := #OCAT OR ("OvercurrentAlarm" AND NOT "AlarmReset");
   "OvercurrentNotify" := #OCAT OR ("OvercurrentNotify" AND NOT "AlarmReset" AND NOT "AlarmSilence");
END_REGION

REGION Network 3
   // High Oil Temp Alarm
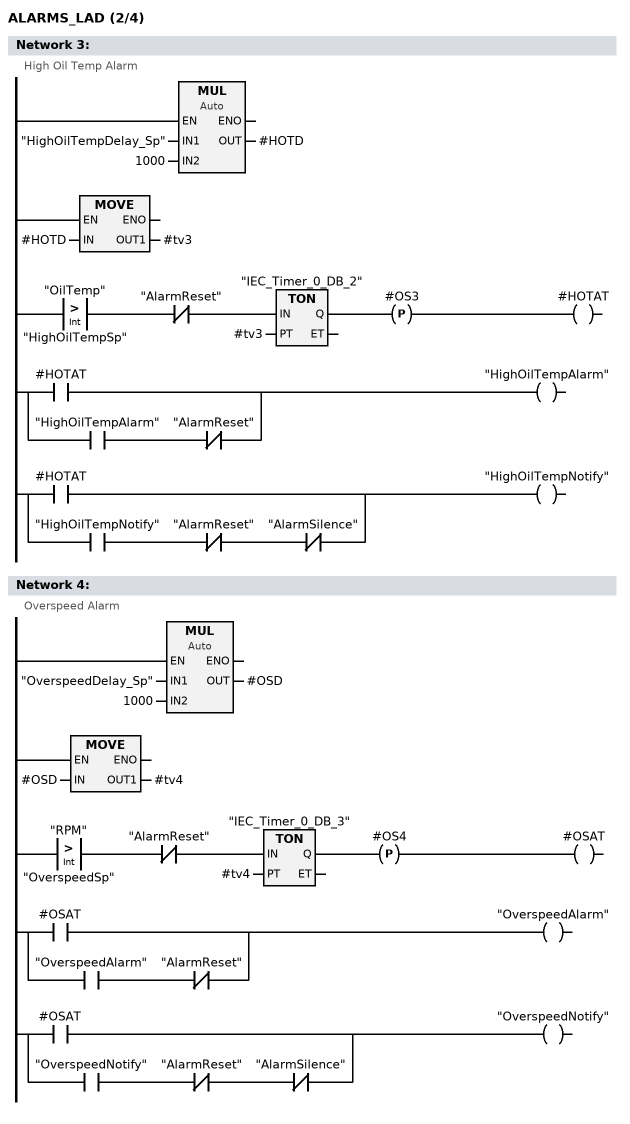
   #HOTD := "HighOilTempDelay_Sp" * 1000;
   #tv3 := #HOTD;
   "IEC_Timer_0_DB_2".TON(IN := ("OilTemp" > "HighOilTempSp") AND NOT "AlarmReset", PT := #tv3);
   #_w1 := "IEC_Timer_0_DB_2".Q AND NOT #OS3;   // rising edge
   #OS3 := "IEC_Timer_0_DB_2".Q;
   #HOTAT := #_w1;
   "HighOilTempAlarm" := #HOTAT OR ("HighOilTempAlarm" AND NOT "AlarmReset");
   "HighOilTempNotify" := #HOTAT OR ("HighOilTempNotify" AND NOT "AlarmReset" AND NOT "AlarmSilence");
END_REGION

REGION Network 4
   // Overspeed Alarm
   #OSD := "OverspeedDelay_Sp" * 1000;
   #tv4 := #OSD;
   "IEC_Timer_0_DB_3".TON(IN := ("RPM" > "OverspeedSp") AND NOT "AlarmReset", PT := #tv4);
   #_w1 := "IEC_Timer_0_DB_3".Q AND NOT #OS4;   // rising edge
   #OS4 := "IEC_Timer_0_DB_3".Q;
   #OSAT := #_w1;
   "OverspeedAlarm" := #OSAT OR ("OverspeedAlarm" AND NOT "AlarmReset");
   "OverspeedNotify" := #OSAT OR ("OverspeedNotify" AND NOT "AlarmReset" AND NOT "AlarmSilence");
END_REGION

REGION Network 5
   // Oil High Flow Alarm
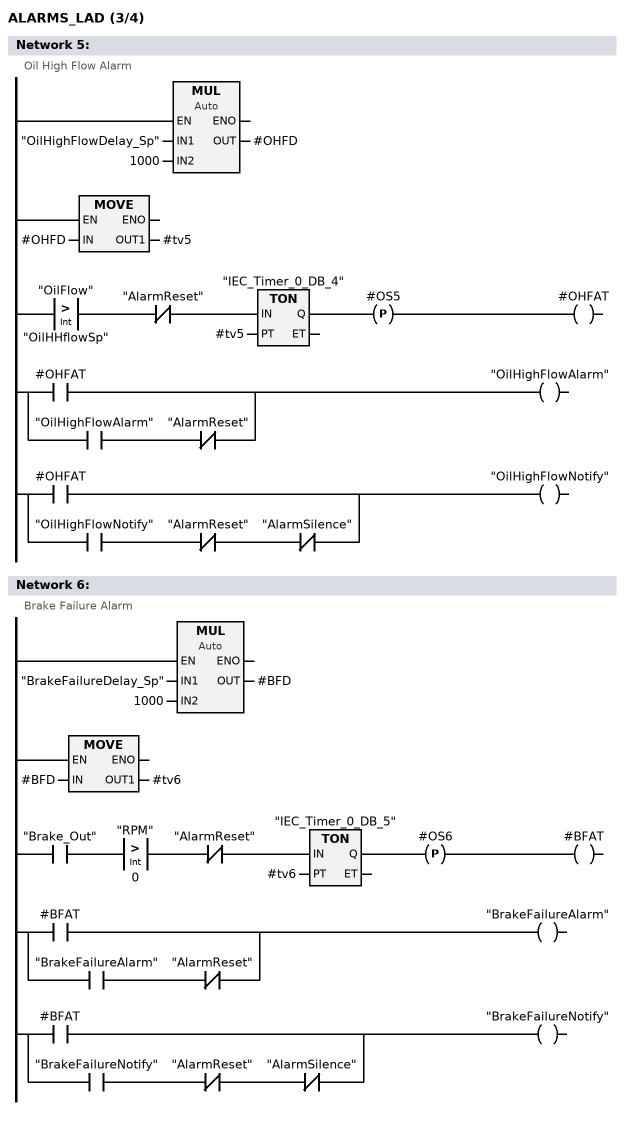
   #OHFD := "OilHighFlowDelay_Sp" * 1000;
   #tv5 := #OHFD;
   "IEC_Timer_0_DB_4".TON(IN := ("OilFlow" > "OilHHflowSp") AND NOT "AlarmReset", PT := #tv5);
   #_w1 := "IEC_Timer_0_DB_4".Q AND NOT #OS5;   // rising edge
   #OS5 := "IEC_Timer_0_DB_4".Q;
   #OHFAT := #_w1;
   "OilHighFlowAlarm" := #OHFAT OR ("OilHighFlowAlarm" AND NOT "AlarmReset");
   "OilHighFlowNotify" := #OHFAT OR ("OilHighFlowNotify" AND NOT "AlarmReset" AND NOT "AlarmSilence");
END_REGION

REGION Network 6
   // Brake Failure Alarm
   #BFD := "BrakeFailureDelay_Sp" * 1000;
   #tv6 := #BFD;
   "IEC_Timer_0_DB_5".TON(IN := "Brake_Out" AND ("RPM" > 0) AND NOT "AlarmReset", PT := #tv6);
   #_w1 := "IEC_Timer_0_DB_5".Q AND NOT #OS6;   // rising edge
   #OS6 := "IEC_Timer_0_DB_5".Q;
   #BFAT := #_w1;
   "BrakeFailureAlarm" := #BFAT OR ("BrakeFailureAlarm" AND NOT "AlarmReset");
   "BrakeFailureNotify" := #BFAT OR ("BrakeFailureNotify" AND NOT "AlarmReset" AND NOT "AlarmSilence");
END_REGION

REGION Network 7
   // EStop Alarm
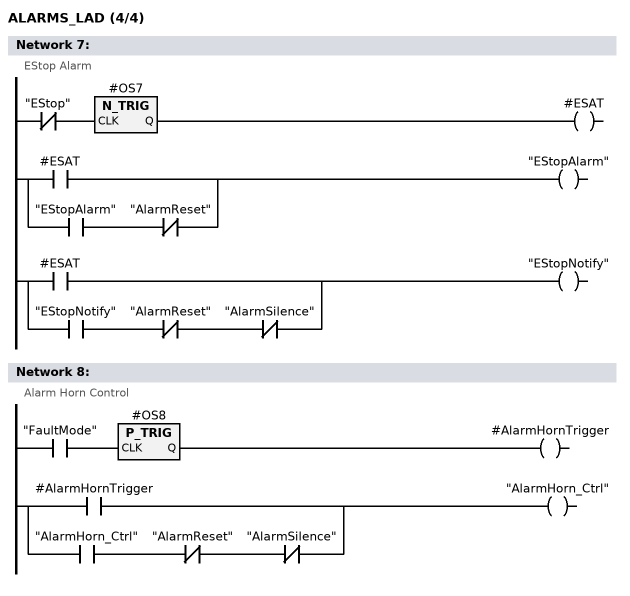
   RUNG wire#powerrail
      I_Contact( "EStop" )
      N_Trig( #OS7 )
      Coil( #ESAT )
   END_RUNG
   RUNG wire#powerrail
      Contact( #ESAT )
      wire#w1
      Coil( "EStopAlarm" )
   END_RUNG
   RUNG wire#powerrail
      Contact( "EStopAlarm" )
      I_Contact( "AlarmReset" )
   END_RUNG wire#w1
   RUNG wire#powerrail
      Contact( #ESAT )
      wire#w2
      Coil( "EStopNotify" )
   END_RUNG
   RUNG wire#powerrail
      Contact( "EStopNotify" )
      I_Contact( "AlarmReset" )
      I_Contact( "AlarmSilence" )
   END_RUNG wire#w2
   // the same network as SCL:
   #_w1 := NOT (NOT "EStop") AND #OS7;   // falling edge
   #OS7 := NOT "EStop";
   #ESAT := #_w1;
   "EStopAlarm" := #ESAT OR ("EStopAlarm" AND NOT "AlarmReset");
   "EStopNotify" := #ESAT OR ("EStopNotify" AND NOT "AlarmReset" AND NOT "AlarmSilence");
END_REGION

REGION Network 8
   // Alarm Horn Control
   RUNG wire#powerrail
      Contact( "FaultMode" )
      P_Trig( #OS8 )
      Coil( #AlarmHornTrigger )
   END_RUNG
   RUNG wire#powerrail
      Contact( #AlarmHornTrigger )
      wire#w1
      Coil( "AlarmHorn_Ctrl" )
   END_RUNG
   RUNG wire#powerrail
      Contact( "AlarmHorn_Ctrl" )
      I_Contact( "AlarmReset" )
      I_Contact( "AlarmSilence" )
   END_RUNG wire#w1
   // the same network as SCL:
   #_w1 := "FaultMode" AND NOT #OS8;   // rising edge
   #OS8 := "FaultMode";
   #AlarmHornTrigger := #_w1;
   "AlarmHorn_Ctrl" := #AlarmHornTrigger OR ("AlarmHorn_Ctrl" AND NOT "AlarmReset" AND NOT "AlarmSilence");
END_REGION
END_FUNCTION_BLOCK

FUNCTION_BLOCK "HOA_FBD"   // FB7, FBD
{ S7_Optimized_Access := 'TRUE' }
VERSION : 0.1
   VAR
      OS1 : Bool;
      OS3 : Bool;
      OS2 : Bool;
      OS4 : Bool;
      OS5 : Bool;
      OS6 : Bool;
      OS7 : Bool;
      OS8 : Bool;
      OS9 : Bool;
      OS10 : Bool;
      OS11 : Bool;
      OS12 : Bool;
   END_VAR
   VAR_TEMP   // added for the SCL form of the ladder/FBD networks
      _w1 : Bool;
      _w2 : Bool;
      _w3 : Bool;
   END_VAR
BEGIN

REGION Network 1
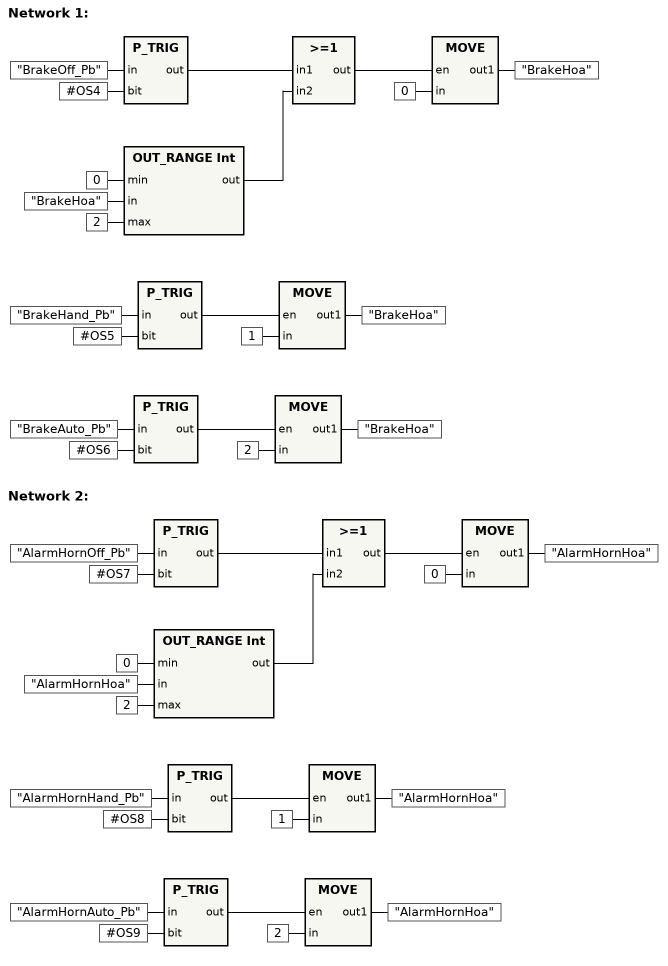
   #_w1 := "BrakeOff_Pb" AND NOT #OS4;   // rising edge
   #OS4 := "BrakeOff_Pb";
   IF #_w1 OR ("BrakeHoa" < 0) OR ("BrakeHoa" > 2) THEN "BrakeHoa" := 0; END_IF;
   #_w2 := "BrakeHand_Pb" AND NOT #OS5;   // rising edge
   #OS5 := "BrakeHand_Pb";
   IF #_w2 THEN "BrakeHoa" := 1; END_IF;
   #_w3 := "BrakeAuto_Pb" AND NOT #OS6;   // rising edge
   #OS6 := "BrakeAuto_Pb";
   IF #_w3 THEN "BrakeHoa" := 2; END_IF;
END_REGION

REGION Network 2
   #_w1 := "AlarmHornOff_Pb" AND NOT #OS7;   // rising edge
   #OS7 := "AlarmHornOff_Pb";
   IF #_w1 OR ("AlarmHornHoa" < 0) OR ("AlarmHornHoa" > 2) THEN "AlarmHornHoa" := 0; END_IF;
   #_w2 := "AlarmHornHand_Pb" AND NOT #OS8;   // rising edge
   #OS8 := "AlarmHornHand_Pb";
   IF #_w2 THEN "AlarmHornHoa" := 1; END_IF;
   #_w3 := "AlarmHornAuto_Pb" AND NOT #OS9;   // rising edge
   #OS9 := "AlarmHornAuto_Pb";
   IF #_w3 THEN "AlarmHornHoa" := 2; END_IF;
END_REGION

REGION Network 3
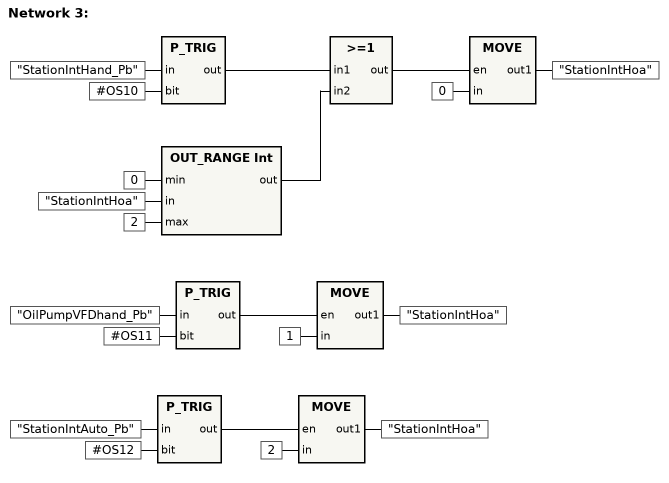
   #_w1 := "StationIntHand_Pb" AND NOT #OS10;   // rising edge
   #OS10 := "StationIntHand_Pb";
   IF #_w1 OR ("StationIntHoa" < 0) OR ("StationIntHoa" > 2) THEN "StationIntHoa" := 0; END_IF;
   #_w2 := "OilPumpVFDhand_Pb" AND NOT #OS11;   // rising edge
   #OS11 := "OilPumpVFDhand_Pb";
   IF #_w2 THEN "StationIntHoa" := 1; END_IF;
   #_w3 := "StationIntAuto_Pb" AND NOT #OS12;   // rising edge
   #OS12 := "StationIntAuto_Pb";
   IF #_w3 THEN "StationIntHoa" := 2; END_IF;
END_REGION
END_FUNCTION_BLOCK

FUNCTION_BLOCK "HOA_LAD"   // FB8, LAD
{ S7_Optimized_Access := 'TRUE' }
VERSION : 0.1
   VAR
      OS1 : Bool;
      OS2 : Bool;
      OS3 : Bool;
      OS4 : Bool;
      OS5 : Bool;
      OS6 : Bool;
      OS7 : Bool;
      OS8 : Bool;
      OS9 : Bool;
      OS10 : Bool;
      OS11 : Bool;
      OS12 : Bool;
   END_VAR
   VAR_TEMP   // added for the SCL form of the ladder/FBD networks
      _w1 : Bool;
      _w2 : Bool;
      _w3 : Bool;
   END_VAR
BEGIN

REGION Network 1
   // // Brake HOA
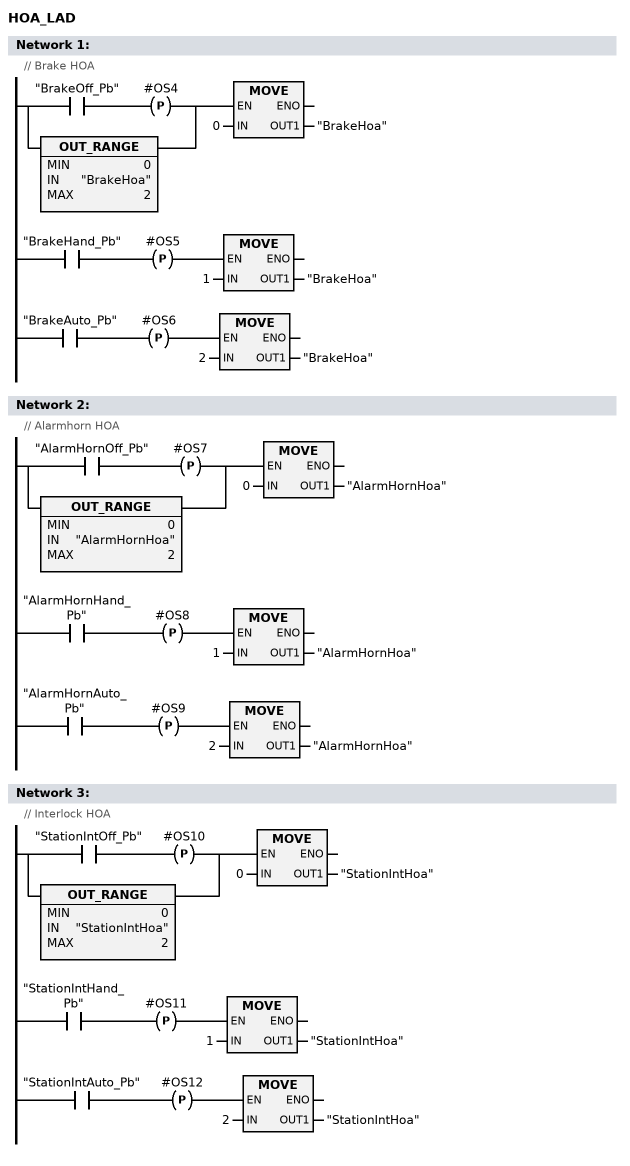
   #_w1 := "BrakeOff_Pb" AND NOT #OS4;   // rising edge
   #OS4 := "BrakeOff_Pb";
   IF #_w1 OR ("BrakeHoa" < 0) OR ("BrakeHoa" > 2) THEN "BrakeHoa" := 0; END_IF;
   #_w2 := "BrakeHand_Pb" AND NOT #OS5;   // rising edge
   #OS5 := "BrakeHand_Pb";
   IF #_w2 THEN "BrakeHoa" := 1; END_IF;
   #_w3 := "BrakeAuto_Pb" AND NOT #OS6;   // rising edge
   #OS6 := "BrakeAuto_Pb";
   IF #_w3 THEN "BrakeHoa" := 2; END_IF;
END_REGION

REGION Network 2
   // // Alarmhorn HOA
   #_w1 := "AlarmHornOff_Pb" AND NOT #OS7;   // rising edge
   #OS7 := "AlarmHornOff_Pb";
   IF #_w1 OR ("AlarmHornHoa" < 0) OR ("AlarmHornHoa" > 2) THEN "AlarmHornHoa" := 0; END_IF;
   #_w2 := "AlarmHornHand_Pb" AND NOT #OS8;   // rising edge
   #OS8 := "AlarmHornHand_Pb";
   IF #_w2 THEN "AlarmHornHoa" := 1; END_IF;
   #_w3 := "AlarmHornAuto_Pb" AND NOT #OS9;   // rising edge
   #OS9 := "AlarmHornAuto_Pb";
   IF #_w3 THEN "AlarmHornHoa" := 2; END_IF;
END_REGION

REGION Network 3
   // // Interlock HOA
   #_w1 := "StationIntOff_Pb" AND NOT #OS10;   // rising edge
   #OS10 := "StationIntOff_Pb";
   IF #_w1 OR ("StationIntHoa" < 0) OR ("StationIntHoa" > 2) THEN "StationIntHoa" := 0; END_IF;
   #_w2 := "StationIntHand_Pb" AND NOT #OS11;   // rising edge
   #OS11 := "StationIntHand_Pb";
   IF #_w2 THEN "StationIntHoa" := 1; END_IF;
   #_w3 := "StationIntAuto_Pb" AND NOT #OS12;   // rising edge
   #OS12 := "StationIntAuto_Pb";
   IF #_w3 THEN "StationIntHoa" := 2; END_IF;
END_REGION
END_FUNCTION_BLOCK

FUNCTION_BLOCK "HOA_SCL"   // FB9, SCL
{ S7_Optimized_Access := 'TRUE' }
VERSION : 0.1
BEGIN
   //Brake HOA Controls
   IF "BrakeHoa" < 0 OR "BrakeHoa" > 2 THEN
       "BrakeHoa" := 0;
   END_IF;

   IF "BrakeOff_Pb" AND "BrakeHoa" <> 0 THEN
       "BrakeHoa" := 0;
   END_IF;

   IF "BrakeHand_Pb" AND "BrakeHoa" <> 1 THEN
       "BrakeHoa" := 1;
   END_IF;

   IF "BrakeAuto_Pb" AND "BrakeHoa" <> 2 THEN
       "BrakeHoa" := 2;
   END_IF;


   //Alarm Horn HOA Controls
   IF "AlarmHornHoa" < 0 OR "AlarmHornHoa" > 2 THEN
       "AlarmHornHoa" := 0;
   END_IF;

   IF "AlarmHornOff_Pb" AND "AlarmHornHoa" <> 0 THEN
       "AlarmHornHoa" := 0;
   END_IF;

   IF "AlarmHornHand_Pb" AND "AlarmHornHoa" <> 1 THEN
       "AlarmHornHoa" := 1;
   END_IF;

   IF "AlarmHornAuto_Pb" AND "AlarmHornHoa" <> 2 THEN
       "AlarmHornHoa" := 2;
   END_IF;


   //Station Interlock HOA Controls
   IF "StationIntHoa" < 0 OR "StationIntHoa" > 2 THEN
       "StationIntHoa" := 0;
   END_IF;

   IF "StationIntOff_Pb" AND "StationIntHoa" <> 0 THEN
       "StationIntHoa" := 0;
   END_IF;

   IF "StationIntHand_Pb" AND "StationIntHoa" <> 1 THEN
       "StationIntHoa" := 1;
   END_IF;

   IF "StationIntAuto_Pb" AND "StationIntHoa" <> 2 THEN
       "StationIntHoa" := 2;
   END_IF;
END_FUNCTION_BLOCK

FUNCTION_BLOCK "HOA_STL"   // FB10, STL
{ S7_Optimized_Access := 'TRUE' }
VERSION : 0.1
   VAR
      OS1 : Bool;
      OS2 : Bool;
      OS4 : Bool;
      OS5 : Bool;
      OS12 : Bool;
      OS6 : Bool;
      OS7 : Bool;
      OS8 : Bool;
      OS9 : Bool;
      OS10 : Bool;
      OS11 : Bool;
      OS3 : Bool;
   END_VAR
BEGIN

REGION Network 1
         L     "BrakeHoa";
         L     0;
         <I;
         JC    SetBrakeHoaZero;
         CLR;
         L     "BrakeHoa";
         L     2;
         >I;
         JC    SetBrakeHoaZero;
         CLR;
         A     "BrakeOff_Pb";
         FP    #OS4;
         JC    SetBrakeHoaZero;
         CLR;
         A     "BrakeHand_Pb";
         FP    #OS5;
         JC    SetBrakeHoaOne;
         CLR;
         A     "BrakeAuto_Pb";
         FP    #OS6;
         JC    SetBrakeHoaTwo;
         JU    AlarmHorn;

   SetBrakeHoaZero:L     0;
         T     "BrakeHoa";
         JU    AlarmHorn;

   SetBrakeHoaOne:L     1;
         T     "BrakeHoa";
         JU    AlarmHorn;

   SetBrakeHoaTwo:L     2;
         T     "BrakeHoa";
         JU    AlarmHorn;


   AlarmHorn:L     "AlarmHornHoa";
         L     0;
         <I;
         JC    SetAlarmHornHoaZero;
         CLR;
         L     "AlarmHornHoa";
         L     2;
         >I;
         JC    SetAlarmHornHoaZero;
         CLR;
         A     "AlarmHornOff_Pb";
         FP    #OS7;
         JC    SetAlarmHornHoaZero;
         CLR;
         A     "AlarmHornHand_Pb";
         FP    #OS8;
         JC    SetBrakeHoaOne;
         CLR;
         A     "AlarmHornAuto_Pb";
         FP    #OS9;
         JC    SetOAlarmHornHoaTwo;
         JU    StationInterlock;

   SetAlarmHornHoaZero:L     0;
         T     "AlarmHornHoa";
         JU    StationInterlock;

   SetOAlarmHornHoaOne:L     1;
         T     "AlarmHornHoa";
         JU    StationInterlock;

   SetOAlarmHornHoaTwo:L     2;
         T     "AlarmHornHoa";
         JU    StationInterlock;


   StationInterlock:L     "StationIntHoa";
         L     0;
         <I;
         JC    SetStationInterlockHoaZero;
         CLR;
         L     "StationIntHoa";
         L     2;
         >I;
         JC    SetStationInterlockHoaZero;
         CLR;
         A     "StationIntOff_Pb";
         FP    #OS10;
         JC    SetStationInterlockHoaZero;
         CLR;
         A     "StationIntHand_Pb";
         FP    #OS11;
         JC    SetStationInterlockHoaOne;
         CLR;
         A     "StationIntAuto_Pb";
         FP    #OS12;
         JC    SetStationInterlockHoaTwo;
         JU    EndOfLine;

   SetStationInterlockHoaZero:L     0;
         T     "StationIntHoa";
         BE;

   SetStationInterlockHoaOne:L     1;
         T     "StationIntHoa";
         BE;

   SetStationInterlockHoaTwo:L     2;
         T     "StationIntHoa";
         BE;

   EndOfLine:BE;
END_REGION
END_FUNCTION_BLOCK

FUNCTION_BLOCK "ALARMS_FBD"   // FB11, FBD
{ S7_Optimized_Access := 'TRUE' }
VERSION : 0.1
   VAR
      OS1 : Bool;
      OS2 : Bool;
      OS3 : Bool;
      OS4 : Bool;
      OS5 : Bool;
      OS6 : Bool;
      OS7 : Bool;
   END_VAR
   VAR_TEMP
      ti1 : Int;
      tt1 : Time;
      ti2 : Int;
      tt2 : Time;
      ti3 : Int;
      tt3 : Time;
      ti4 : Int;
      tt4 : Time;
      ti5 : Int;
      tt5 : Time;
      ti6 : Int;
      tt6 : Time;
   END_VAR
   VAR_TEMP   // added for the SCL form of the ladder/FBD networks
      _w1 : Bool;
   END_VAR
BEGIN

REGION Network 1
   // Oil Low Flow Alarm
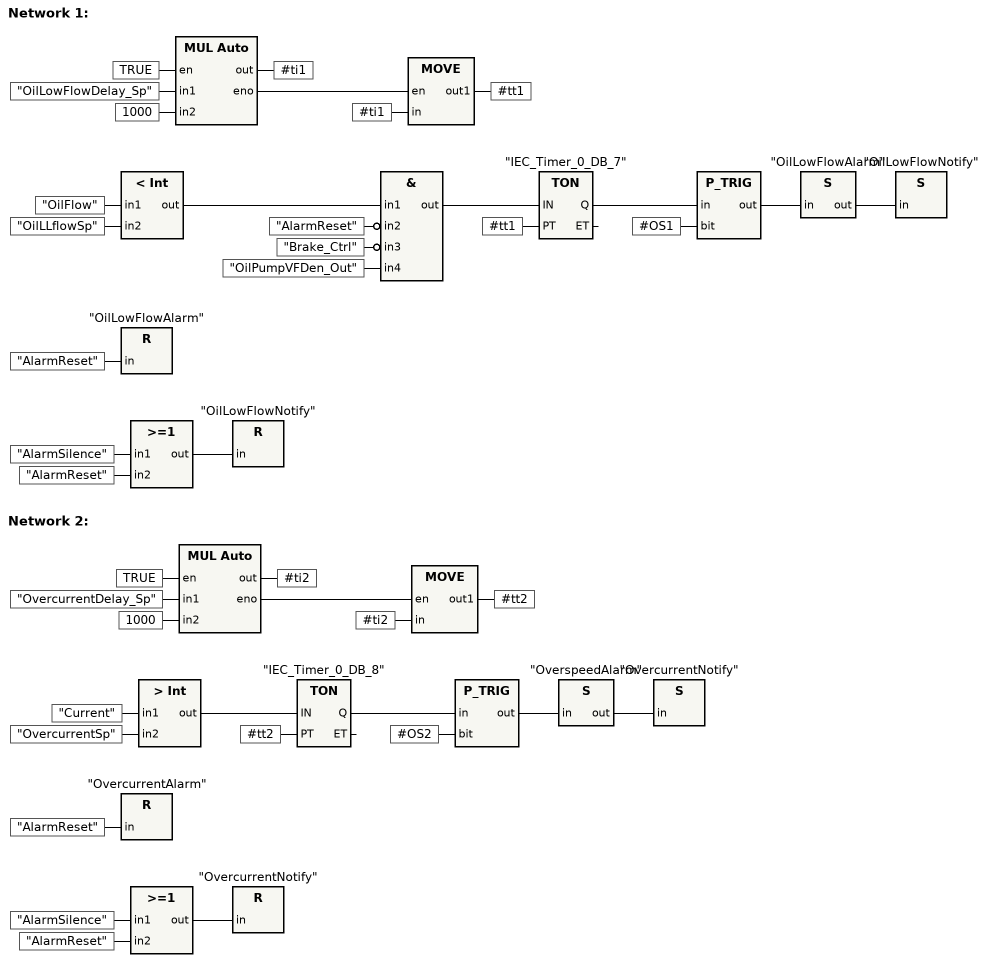
   IF TRUE THEN
       #ti1 := "OilLowFlowDelay_Sp" * 1000;
       #tt1 := #ti1;
   END_IF;
   "IEC_Timer_0_DB_7".TON(IN := ("OilFlow" < "OilLLflowSp") AND NOT "AlarmReset" AND NOT "Brake_Ctrl" AND "OilPumpVFDen_Out",
                          PT := #tt1);
   #_w1 := "IEC_Timer_0_DB_7".Q AND NOT #OS1;   // rising edge
   #OS1 := "IEC_Timer_0_DB_7".Q;
   IF #_w1 THEN
       "OilLowFlowAlarm" := TRUE;
       "OilLowFlowNotify" := TRUE;
   END_IF;
   IF "AlarmReset" THEN "OilLowFlowAlarm" := FALSE; END_IF;
   IF "AlarmSilence" OR "AlarmReset" THEN "OilLowFlowNotify" := FALSE; END_IF;
END_REGION

REGION Network 2
   // Overcurrent Alarm
   IF TRUE THEN
       #ti2 := "OvercurrentDelay_Sp" * 1000;
       #tt2 := #ti2;
   END_IF;
   "IEC_Timer_0_DB_8".TON(IN := "Current" > "OvercurrentSp", PT := #tt2);
   #_w1 := "IEC_Timer_0_DB_8".Q AND NOT #OS2;   // rising edge
   #OS2 := "IEC_Timer_0_DB_8".Q;
   IF #_w1 THEN
       "OverspeedAlarm" := TRUE;
       "OvercurrentNotify" := TRUE;
   END_IF;
   IF "AlarmReset" THEN "OvercurrentAlarm" := FALSE; END_IF;
   IF "AlarmSilence" OR "AlarmReset" THEN "OvercurrentNotify" := FALSE; END_IF;
END_REGION

REGION Network 3
   // High Oil Temp Alarm
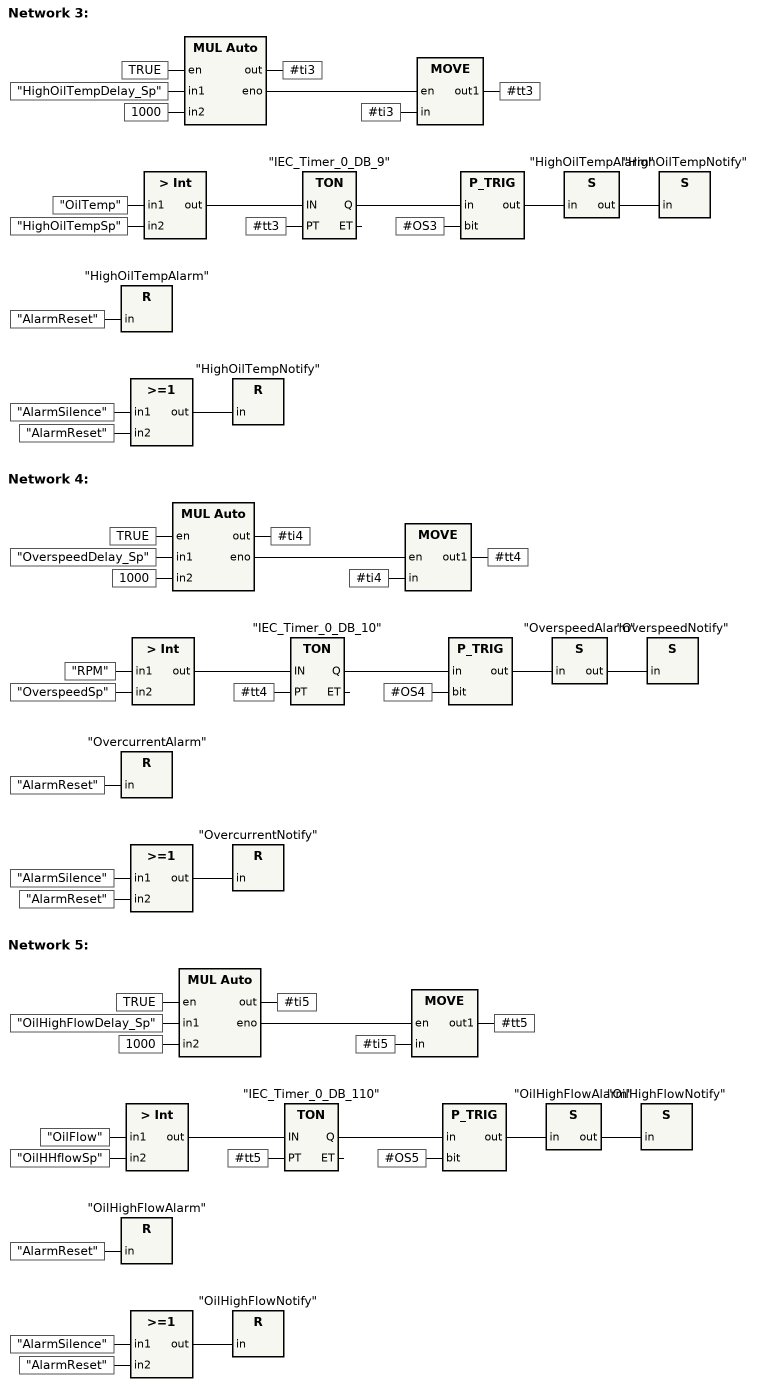
   IF TRUE THEN
       #ti3 := "HighOilTempDelay_Sp" * 1000;
       #tt3 := #ti3;
   END_IF;
   "IEC_Timer_0_DB_9".TON(IN := "OilTemp" > "HighOilTempSp", PT := #tt3);
   #_w1 := "IEC_Timer_0_DB_9".Q AND NOT #OS3;   // rising edge
   #OS3 := "IEC_Timer_0_DB_9".Q;
   IF #_w1 THEN
       "HighOilTempAlarm" := TRUE;
       "HighOilTempNotify" := TRUE;
   END_IF;
   IF "AlarmReset" THEN "HighOilTempAlarm" := FALSE; END_IF;
   IF "AlarmSilence" OR "AlarmReset" THEN "HighOilTempNotify" := FALSE; END_IF;
END_REGION

REGION Network 4
   // Overspeed Alarm
   IF TRUE THEN
       #ti4 := "OverspeedDelay_Sp" * 1000;
       #tt4 := #ti4;
   END_IF;
   "IEC_Timer_0_DB_10".TON(IN := "RPM" > "OverspeedSp", PT := #tt4);
   #_w1 := "IEC_Timer_0_DB_10".Q AND NOT #OS4;   // rising edge
   #OS4 := "IEC_Timer_0_DB_10".Q;
   IF #_w1 THEN
       "OverspeedAlarm" := TRUE;
       "OverspeedNotify" := TRUE;
   END_IF;
   IF "AlarmReset" THEN "OvercurrentAlarm" := FALSE; END_IF;
   IF "AlarmSilence" OR "AlarmReset" THEN "OvercurrentNotify" := FALSE; END_IF;
END_REGION

REGION Network 5
   // High Oil Flow Alarm
   IF TRUE THEN
       #ti5 := "OilHighFlowDelay_Sp" * 1000;
       #tt5 := #ti5;
   END_IF;
   "IEC_Timer_0_DB_110".TON(IN := "OilFlow" > "OilHHflowSp", PT := #tt5);
   #_w1 := "IEC_Timer_0_DB_110".Q AND NOT #OS5;   // rising edge
   #OS5 := "IEC_Timer_0_DB_110".Q;
   IF #_w1 THEN
       "OilHighFlowAlarm" := TRUE;
       "OilHighFlowNotify" := TRUE;
   END_IF;
   IF "AlarmReset" THEN "OilHighFlowAlarm" := FALSE; END_IF;
   IF "AlarmSilence" OR "AlarmReset" THEN "OilHighFlowNotify" := FALSE; END_IF;
END_REGION

REGION Network 6
   // Brake Failure Alarm
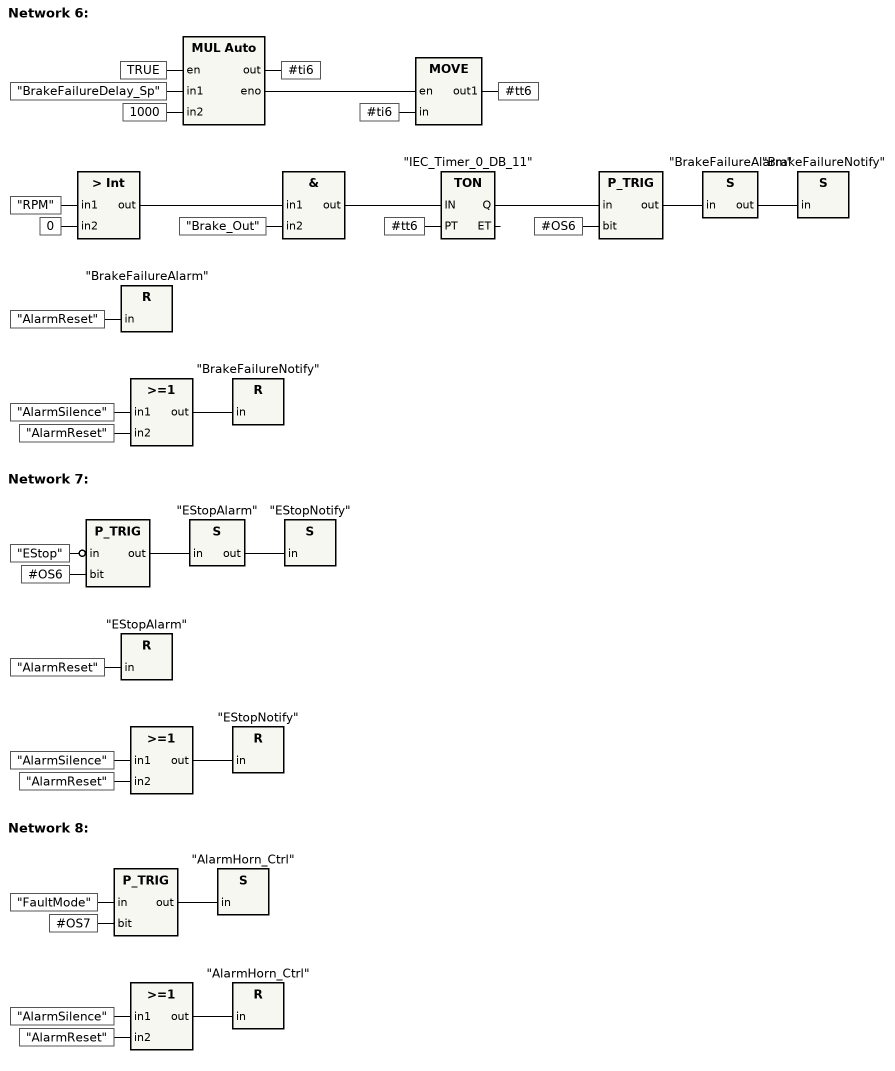
   IF TRUE THEN
       #ti6 := "BrakeFailureDelay_Sp" * 1000;
       #tt6 := #ti6;
   END_IF;
   "IEC_Timer_0_DB_11".TON(IN := ("RPM" > 0) AND "Brake_Out", PT := #tt6);
   #_w1 := "IEC_Timer_0_DB_11".Q AND NOT #OS6;   // rising edge
   #OS6 := "IEC_Timer_0_DB_11".Q;
   IF #_w1 THEN
       "BrakeFailureAlarm" := TRUE;
       "BrakeFailureNotify" := TRUE;
   END_IF;
   IF "AlarmReset" THEN "BrakeFailureAlarm" := FALSE; END_IF;
   IF "AlarmSilence" OR "AlarmReset" THEN "BrakeFailureNotify" := FALSE; END_IF;
END_REGION

REGION Network 7
   // EStop Alarm
   #_w1 := NOT "EStop" AND NOT #OS6;   // rising edge
   #OS6 := NOT "EStop";
   IF #_w1 THEN
       "EStopAlarm" := TRUE;
       "EStopNotify" := TRUE;
   END_IF;
   IF "AlarmReset" THEN "EStopAlarm" := FALSE; END_IF;
   IF "AlarmSilence" OR "AlarmReset" THEN "EStopNotify" := FALSE; END_IF;
END_REGION

REGION Network 8
   // Alarm Horn Control
   #_w1 := "FaultMode" AND NOT #OS7;   // rising edge
   #OS7 := "FaultMode";
   IF #_w1 THEN "AlarmHorn_Ctrl" := TRUE; END_IF;
   IF "AlarmSilence" OR "AlarmReset" THEN "AlarmHorn_Ctrl" := FALSE; END_IF;
END_REGION
END_FUNCTION_BLOCK

FUNCTION_BLOCK "ALARMS_SCL"   // FB12, SCL
{ S7_Optimized_Access := 'TRUE' }
VERSION : 0.1
   VAR_TEMP
      ti1 : Time;
      LOFAT : Bool;
      t1 : Time;
      ti2 : Time;
      ti3 : Time;
      ti4 : Time;
      ti5 : Time;
      ti6 : Time;
      ti7 : Time;
      t2 : Time;
      t3 : Time;
      t4 : Time;
      t5 : Time;
      t6 : Time;
      t7 : Time;
      OCAT : Bool;
      HOTAT : Bool;
      OSAT : Bool;
      HOFAT : Bool;
      BFAT : Bool;
   END_VAR
BEGIN
   //Oil Low Flow Alarm
   IF "OilPumpVFDen_Out" AND "OilFlow" < "OilLLflowSp" AND NOT "Brake_Out" AND NOT "OilLowFlowAlarm" AND NOT "AlarmReset" THEN
       "CONVERTTIME"(Int1 := "OilLowFlowDelay_Sp",
                     Time1 => #ti1);

       "IEC_Timer_0_DB_12".TON(IN := TRUE,
                               PT := #ti1,
                               Q => #LOFAT,
                               ET => #t1);
   END_IF;

   IF #LOFAT THEN
       "OilLowFlowAlarm" := 1;
       "OilLowFlowNotify" := 1;
   END_IF;

   IF "OilLowFlowAlarm" AND "AlarmReset" THEN
       "OilLowFlowAlarm" := 0;
       "OilLowFlowNotify" := 0;
   END_IF;

   IF "OilLowFlowNotify" AND "AlarmSilence" THEN
       "OilLowFlowNotify" := 0;
   END_IF;



   //Overcurrent Alarm
   IF "Current" > "OvercurrentSp" AND NOT "OvercurrentAlarm" AND NOT "AlarmReset" THEN
       "CONVERTTIME"(Int1:="OvercurrentDelay_Sp",
                     Time1=>#ti2);

       "IEC_Timer_0_DB_13".TON(IN:=TRUE,
                           PT:=#ti2,
                           Q=>#OCAT,
                           ET=>#t2);
   END_IF;

   IF #OCAT THEN
       "OvercurrentAlarm" := 1;
       "OvercurrentNotify" := 1;
   END_IF;

   IF "OvercurrentAlarm" AND "AlarmReset" THEN
       "OvercurrentAlarm" := 0;
       "OvercurrentNotify" := 0;
   END_IF;

   IF "OvercurrentNotify" AND "AlarmSilence" THEN
       "OvercurrentNotify" := 0;
   END_IF;




   //High Oil Temp Alarm
   IF "OilTemp" > "HighOilTempSp" AND NOT "HighOilTempAlarm" AND NOT "AlarmReset" THEN
       "CONVERTTIME"(Int1 := "HighOilTempDelay_Sp",
                     Time1 => #ti3);

   "IEC_Timer_0_DB_14".TON(IN:=TRUE,
                           PT:=#ti3,
                           Q=>#HOTAT,
                           ET=>#t3);
   END_IF;

   IF #HOTAT THEN
       "HighOilTempAlarm" := 1;
       "HighOilTempNotify" := 1;
   END_IF;

   IF "HighOilTempAlarm" AND "AlarmReset" THEN
       "HighOilTempAlarm" := 0;
       "HighOilTempNotify" := 0;
   END_IF;

   IF "HighOilTempNotify" AND "AlarmSilence" THEN
       "HighOilTempNotify" := 0;
   END_IF;



   //Overspeed Alarm
   IF "RPM" > "OverspeedSp" AND NOT "OverspeedAlarm" AND NOT "AlarmReset" THEN
   "CONVERTTIME"(Int1:="OverspeedDelay_Sp",
                 Time1=>#ti4);
   "IEC_Timer_0_DB_15".TON(IN:=TRUE,
                           PT:=#ti4,
                           Q=>#OSAT,
                           ET=>#t4);
   END_IF;

   IF #OSAT THEN
       "OverspeedAlarm" := 1;
       "OverspeedNotify" := 1;
   END_IF;

   IF "OverspeedAlarm" AND "AlarmReset" THEN
       "OverspeedAlarm" := 0;
       "OverspeedNotify" := 0;
   END_IF;

   IF "OverspeedNotify" AND "AlarmSilence" THEN
       "OverspeedNotify" := 0;
   END_IF;



   //High Oil Flow Alarm
   IF "OilFlow" > "OilHHflowSp" AND NOT "OilHighFlowAlarm" AND NOT "AlarmReset" THEN
   "CONVERTTIME"(Int1:="OilHighFlowDelay_Sp",
                 Time1=>#ti5);
   "IEC_Timer_0_DB_16".TON(IN:=TRUE,
                           PT:=#ti5,
                           Q=>#HOFAT,
                           ET=>#t5);

   END_IF;

   IF #HOFAT THEN
       "OilHighFlowAlarm" := 1;
       "OilHighFlowNotify" := 1;
   END_IF;

   IF "OilHighFlowAlarm" AND "AlarmReset" THEN
       "OilHighFlowAlarm" := 0;
       "OilHighFlowNotify" := 0;
   END_IF;

   IF "OilHighFlowNotify" AND "AlarmSilence" THEN
       "OilHighFlowNotify" := 0;
   END_IF;



   //Brake Failure Alarm
   IF "Brake_Out" AND "RPM" > 0 AND NOT "BrakeFailureAlarm" AND NOT "AlarmReset" THEN
   "CONVERTTIME"(Int1:="BrakeFailureDelay_Sp",
                 Time1=>#ti6);
   "IEC_Timer_0_DB_17".TON(IN:=TRUE,
                           PT:=#ti6,
                           Q=>#BFAT,
                           ET=>#t6);
   END_IF;

   IF #BFAT THEN
       "BrakeFailureAlarm" := 1;
       "BrakeFailureNotify" := 1;
   END_IF;

   IF "BrakeFailureAlarm" AND "AlarmReset" THEN
       "BrakeFailureAlarm" := 0;
       "BrakeFailureNotify" := 0;
   END_IF;

   IF "BrakeFailureNotify" AND "AlarmSilence" THEN
       "BrakeFailureNotify" := 0;
   END_IF;



   //EStop Alarm
   IF NOT "EStop" AND NOT "EStopAlarm" THEN
       "EStopAlarm" := 1;
       "EStopNotify" := 1;
   END_IF;

   IF "EStopAlarm" AND "AlarmReset" THEN
       "EStopAlarm" := 0;
       "EStopNotify" := 0;
   END_IF;

   IF "EStopNotify" AND "AlarmSilence" THEN
       "EStopNotify" := 0;
   END_IF;



   //Alarm Horn Control
   IF "FaultMode" AND NOT "AlarmHorn_Ctrl" THEN
       "AlarmHorn_Ctrl" := 1;
   END_IF;

   IF "AlarmHorn_Ctrl" AND ("AlarmReset" OR "AlarmSilence") THEN
       "AlarmHorn_Ctrl" := 0;
   END_IF;
END_FUNCTION_BLOCK

FUNCTION_BLOCK "ALARMS_STL"   // FB13, STL
{ S7_Optimized_Access := 'TRUE' }
VERSION : 0.1
   VAR
      OS1 : Bool;
      OS2 : Bool;
      OS3 : Bool;
      OS4 : Bool;
      OS5 : Bool;
      OS6 : Bool;
      OS7 : Bool;
      OS8 : Bool;
      OS9 : Bool;
      OS10 : Bool;
      OS11 : Bool;
      OS12 : Bool;
      OS13 : Bool;
      OS14 : Bool;
      OS15 : Bool;
      OS16 : Bool;
      OS17 : Bool;
   END_VAR
   VAR_TEMP
      ti1 : Time;
      ti2 : Time;
      ti3 : Time;
      ti4 : Time;
      ti5 : Time;
      ti6 : Time;
      ti7 : Time;
      t1 : Time;
      t2 : Time;
      t3 : Time;
      t4 : Time;
      t5 : Time;
      t6 : Time;
      t7 : Time;
      OILAT : Bool;
      OLFAT : Bool;
      OCAT : Bool;
      HOTAT : Bool;
      OSAT : Bool;
      HOFAT : Bool;
      BFAT : Bool;
   END_VAR
BEGIN

REGION Network 1
   //Oil Low Flow Alarm
         L     "OilFlow";
         L     "OilLLflowSp";
         <I;
         A     "OilPumpVFDen_Out";
         AN    "Brake_Out";
         JC    OLFtimer;
         CLR;
         A     "AlarmReset";
         FP    #OS1;
         JC    ResetOLFalarm;
         CLR;
         A     "AlarmSilence";
         FP    #OS2;
         JC    ResetOLFnotify;
         JU    OvercurrentAlarm;

   OLFtimer:CALL  "CONVERTTIME"
         ( Int1  := "OilLowFlowDelay_Sp",
           Time1 := #ti1
         );
         CALL  TON, "IEC_Timer_0_DB_18"
         ( IN := TRUE,
           PT := #ti1,
           Q  := #OLFAT,
           ET := #t1
         );
         A     #OLFAT;
         JC    SetOLFalarm;
         JU    OvercurrentAlarm;

   SetOLFalarm:SET;
         S     "OilLowFlowAlarm";
         S     "OilLowFlowNotify";
         JU    OvercurrentAlarm;

   ResetOLFalarm:R     "OilLowFlowAlarm";
         R     "OilLowFlowNotify";
         JU    OvercurrentAlarm;

   ResetOLFnotify:R     "OilLowFlowNotify";
         JU    OvercurrentAlarm;


   //Overcurrent Alarm
   OvercurrentAlarm:L     "Current";
         L     "OvercurrentSp";
         >I;
         JC    OCtimer;
         CLR;
         A     "AlarmReset";
         FP    #OS3;
         JC    ResetOCalarm;
         CLR;
         A     "AlarmSilence";
         FP    #OS4;
         JC    ResetOCnotify;
         JU    HighOilTempAlarm;

   OCtimer:CALL  "CONVERTTIME"
         ( Int1  := "OvercurrentDelay_Sp",
           Time1 := #ti2
         );
         CALL  TON, "IEC_Timer_0_DB_19"
         ( IN := true,
           PT := #ti2,
           Q  := #OCAT,
           ET := #t2
         );
         A     #OCAT;
         JC    SetOCalarm;
         JU    HighOilTempAlarm;

   SetOCalarm:SET;
         S     "OvercurrentAlarm";
         S     "OvercurrentNotify";
         JU    HighOilTempAlarm;

   ResetOCalarm:R     "OvercurrentAlarm";
         R     "OvercurrentNotify";
         JU    HighOilTempAlarm;

   ResetOCnotify:R     "OvercurrentNotify";
         JU    HighOilTempAlarm;


   //High Oil Temp Alarm
   HighOilTempAlarm:L     "OilTemp";
         L     "HighOilTempSp";
         >I;
         JC    HOTtimer;
         CLR;
         A     "AlarmReset";
         FP    #OS5;
         JC    ResetHOTalarm;
         CLR;
         A     "AlarmSilence";
         FP    #OS6;
         JC    ResetHOTnotify;
         JU    OverspeedAlarm;

   HOTtimer:CALL  "CONVERTTIME"
         ( Int1  := "HighOilTempDelay_Sp",
           Time1 := #ti3
         );
         CALL  TON, "IEC_Timer_0_DB_20"
         ( IN := TRUE,
           PT := #ti3,
           Q  := #HOTAT,
           ET := #t3
         );
         A     #HOTAT;
         JC    SetHOTalarm;
         JU    OverspeedAlarm;

   SetHOTalarm:SET;
         S     "HighOilTempAlarm";
         S     "HighOilTempNotify";
         JU    OverspeedAlarm;

   ResetHOTalarm:R     "HighOilTempAlarm";
         R     "HighOilTempNotify";
         JU    OverspeedAlarm;

   ResetHOTnotify:R     "HighOilTempNotify";
         JU    OverspeedAlarm;


   //Overspeed Alarm
   OverspeedAlarm:L     "RPM";
         L     "OverspeedSp";
         >I;
         JC    OStimer;
         CLR;
         A     "AlarmReset";
         FP    #OS7;
         JC    ResetOSalarm;
         CLR;
         A     "AlarmSilence";
         FP    #OS8;
         JC    ResetOSnotify;
         JU    HighOilFlowAlarm;

   OStimer:CALL  "CONVERTTIME"
         ( Int1  := "OverspeedDelay_Sp",
           Time1 := #ti4
         );
         CALL  TON, "IEC_Timer_0_DB_21"
         ( IN := TRUE,
           PT := #ti4,
           Q  := #OSAT,
           ET := #t4
         );
         A     #OSAT;
         JC    SetOSalarm;
         JU    HighOilFlowAlarm;

   SetOSalarm:SET;
         S     "OverspeedAlarm";
         S     "OverspeedNotify";
         JU    HighOilFlowAlarm;

   ResetOSalarm:R     "OverspeedAlarm";
         R     "OverspeedNotify";
         JU    HighOilFlowAlarm;

   ResetOSnotify:R     "OverspeedNotify";
         JU    HighOilFlowAlarm;


   //High Oil Flow Alarm
   HighOilFlowAlarm:L     "OilFlow";
         L     "OilHHflowSp";
         >I;
         JC    HOFtimer;
         CLR;
         A     "AlarmReset";
         FP    #OS9;
         JC    ResetHOFalarm;
         CLR;
         A     "AlarmSilence";
         FP    #OS10;
         JC    ResetHOFnotify;
         JU    BrakeFailureAlarm;

   HOFtimer:CALL  "CONVERTTIME"
         ( Int1  := "OilHighFlowDelay_Sp",
           Time1 := #ti5
         );
         CALL  TON, "IEC_Timer_0_DB_22"
         ( IN := TRUE,
           PT := #ti5,
           Q  := #HOFAT,
           ET := #t5
         );
         A     #HOFAT;
         JC    SetHOFalarm;
         JU    BrakeFailureAlarm;

   SetHOFalarm:SET;
         S     "OilHighFlowAlarm";
         S     "OilHighFlowNotify";
         JU    BrakeFailureAlarm;

   ResetHOFalarm:R     "OilHighFlowAlarm";
         R     "OilHighFlowNotify";
         JU    BrakeFailureAlarm;

   ResetHOFnotify:R     "OilHighFlowNotify";
         JU    BrakeFailureAlarm;


   //Brake Failure Alarm
   BrakeFailureAlarm:L     "RPM";
         L     0;
         >I;
         A     "Brake_Out";
         JC    BFtimer;
         CLR;
         A     "AlarmReset";
         FP    #OS11;
         JC    ResetBFalarm;
         CLR;
         A     "AlarmSilence";
         FP    #OS12;
         JC    ResetBFnotify;
         JU    EStoplarm;

   BFtimer:CALL  "CONVERTTIME"
         ( Int1  := "BrakeFailureDelay_Sp",
           Time1 := #ti6
         );
         CALL  TON, "IEC_Timer_0_DB_23"
         ( IN := TRUE,
           PT := #ti6,
           Q  := #BFAT,
           ET :=
         );
         A     #BFAT;
         JC    SetBFalarm;
         JU    EStoplarm;

   SetBFalarm:SET;
         S     "BrakeFailureAlarm";
         S     "BrakeFailureNotify";
         JU    EStoplarm;

   ResetBFalarm:R     "BrakeFailureAlarm";
         R     "BrakeFailureNotify";
         JU    EStoplarm;

   ResetBFnotify:R     "BrakeFailureNotify";
         JU    EStoplarm;


   //EStop Alarm
   EStoplarm:AN    "EStop";
         FP    #OS13;
         JC    SetESalarm;
         CLR;
         A     "AlarmReset";
         FP    #OS14;
         JC    ResetESalarm;
         CLR;
         A     "AlarmSilence";
         FP    #OS15;
         JC    ResetESnotify;
         JU    AlarmHornCtrl;

   SetESalarm:SET;
         S     "EStopAlarm";
         S     "EStopNotify";
         JU    AlarmHornCtrl;

   ResetESalarm:R     "EStopAlarm";
         R     "EStopNotify";
         JU    AlarmHornCtrl;

   ResetESnotify:R     "EStopNotify";
         JU    AlarmHornCtrl;



   //Alarm Horn Control
   AlarmHornCtrl:A     "FaultMode";
         FP    #OS16;
         JC    SetAlarmHorn;
         CLR;
         A     "AlarmReset";
         O     "AlarmSilence";
         FP    #OS17;
         JC    ResetAlarmHorn;
         JU    EndOfLine;

   SetAlarmHorn:SET;
         S     "AlarmHorn_Ctrl";
         JU    EndOfLine;

   ResetAlarmHorn:R     "AlarmHorn_Ctrl";
         JU    EndOfLine;



   EndOfLine:BE;
END_REGION
END_FUNCTION_BLOCK

FUNCTION_BLOCK "MODES_LAD"   // FB14, LAD
{ S7_Optimized_Access := 'TRUE' }
VERSION : 0.1
   VAR
      OS1 : Bool;
      OS2 : Bool;
      OS3 : Bool;
      OS4 : Bool;
      OS5 : Bool;
   END_VAR
   VAR_TEMP
      tv1 : Int;
      ti1 : Time;
      tv2 : Int;
      tv3 : Int;
      tv4 : Int;
      ti2 : Time;
      tv5 : Int;
      ti3 : Time;
   END_VAR
   VAR_TEMP   // added for the SCL form of the ladder/FBD networks
      _w1 : Bool;
      _w2 : Bool;
      _w3 : Bool;
   END_VAR
BEGIN

REGION Network 1
   // Warmup Mode
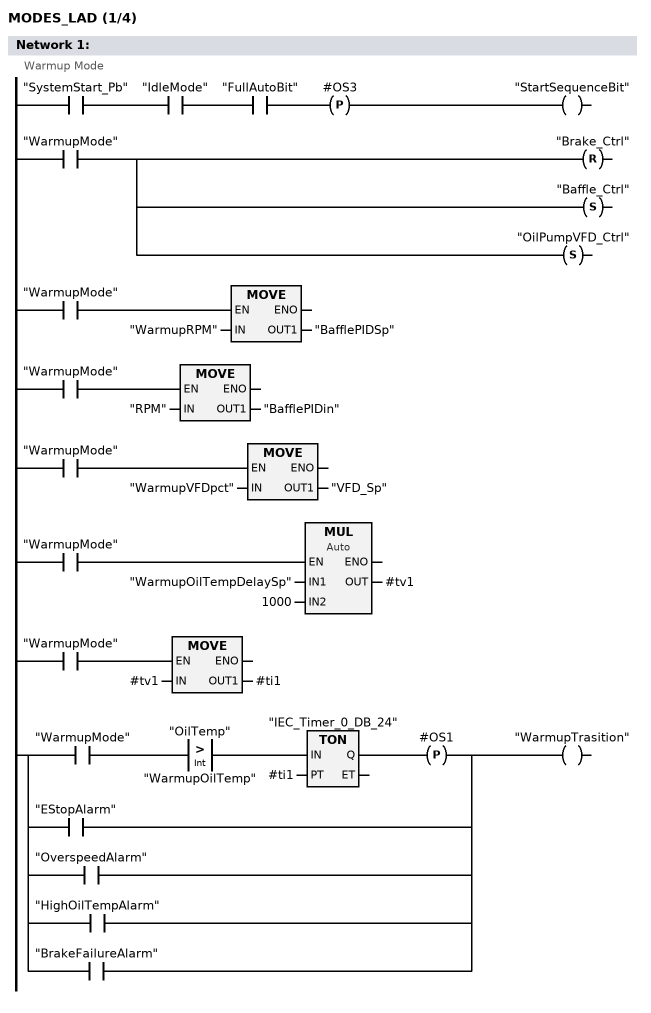
   #_w1 := "SystemStart_Pb" AND "IdleMode" AND "FullAutoBit";
   #_w2 := #_w1 AND NOT #OS3;   // rising edge
   #OS3 := #_w1;
   "StartSequenceBit" := #_w2;
   IF "WarmupMode" THEN
       "Brake_Ctrl" := FALSE;
       "Baffle_Ctrl" := TRUE;
       "OilPumpVFD_Ctrl" := TRUE;
       "BafflePIDSp" := "WarmupRPM";
       "BafflePIDin" := "RPM";
       "VFD_Sp" := "WarmupVFDpct";
       #tv1 := "WarmupOilTempDelaySp" * 1000;
       #ti1 := #tv1;
   END_IF;
   "IEC_Timer_0_DB_24".TON(IN := "WarmupMode" AND ("OilTemp" > "WarmupOilTemp"), PT := #ti1);
   #_w3 := "IEC_Timer_0_DB_24".Q AND NOT #OS1;   // rising edge
   #OS1 := "IEC_Timer_0_DB_24".Q;
   "WarmupTrasition" := #_w3 OR "EStopAlarm" OR "OverspeedAlarm" OR "HighOilTempAlarm" OR "BrakeFailureAlarm";
END_REGION

REGION Network 2
   // Stabilize Mode
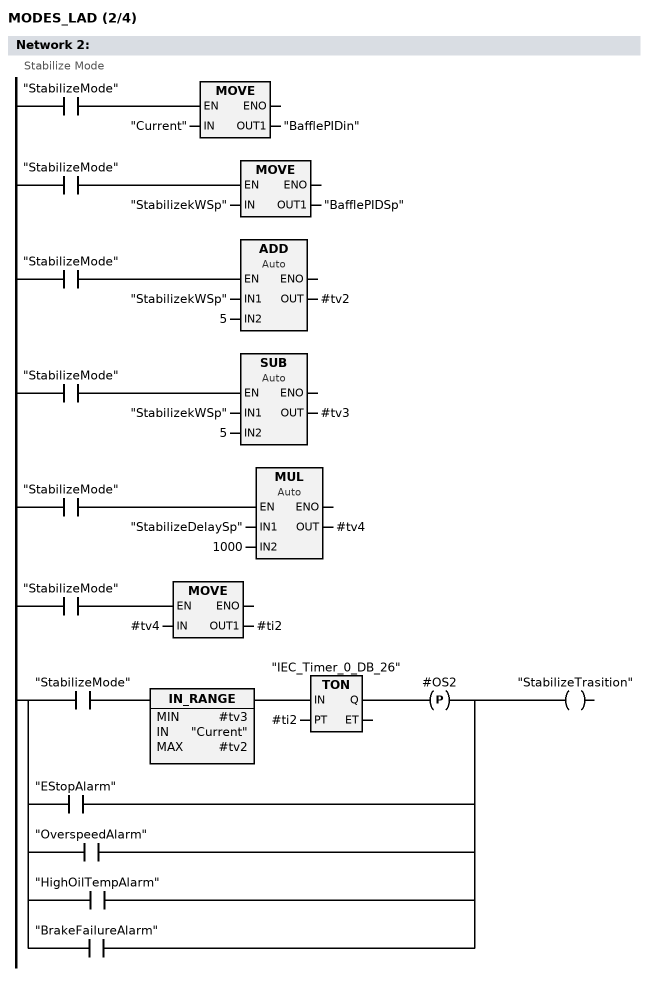
   IF "StabilizeMode" THEN
       "BafflePIDin" := "Current";
       "BafflePIDSp" := "StabilizekWSp";
       #tv2 := "StabilizekWSp" + 5;
       #tv3 := "StabilizekWSp" - 5;
       #tv4 := "StabilizeDelaySp" * 1000;
       #ti2 := #tv4;
   END_IF;
   "IEC_Timer_0_DB_26".TON(IN := "StabilizeMode" AND (#tv3 <= "Current") AND ("Current" <= #tv2), PT := #ti2);
   #_w1 := "IEC_Timer_0_DB_26".Q AND NOT #OS2;   // rising edge
   #OS2 := "IEC_Timer_0_DB_26".Q;
   "StabilizeTrasition" := #_w1 OR "EStopAlarm" OR "OverspeedAlarm" OR "HighOilTempAlarm" OR "BrakeFailureAlarm";
END_REGION

REGION Network 3
   // Generation Mode
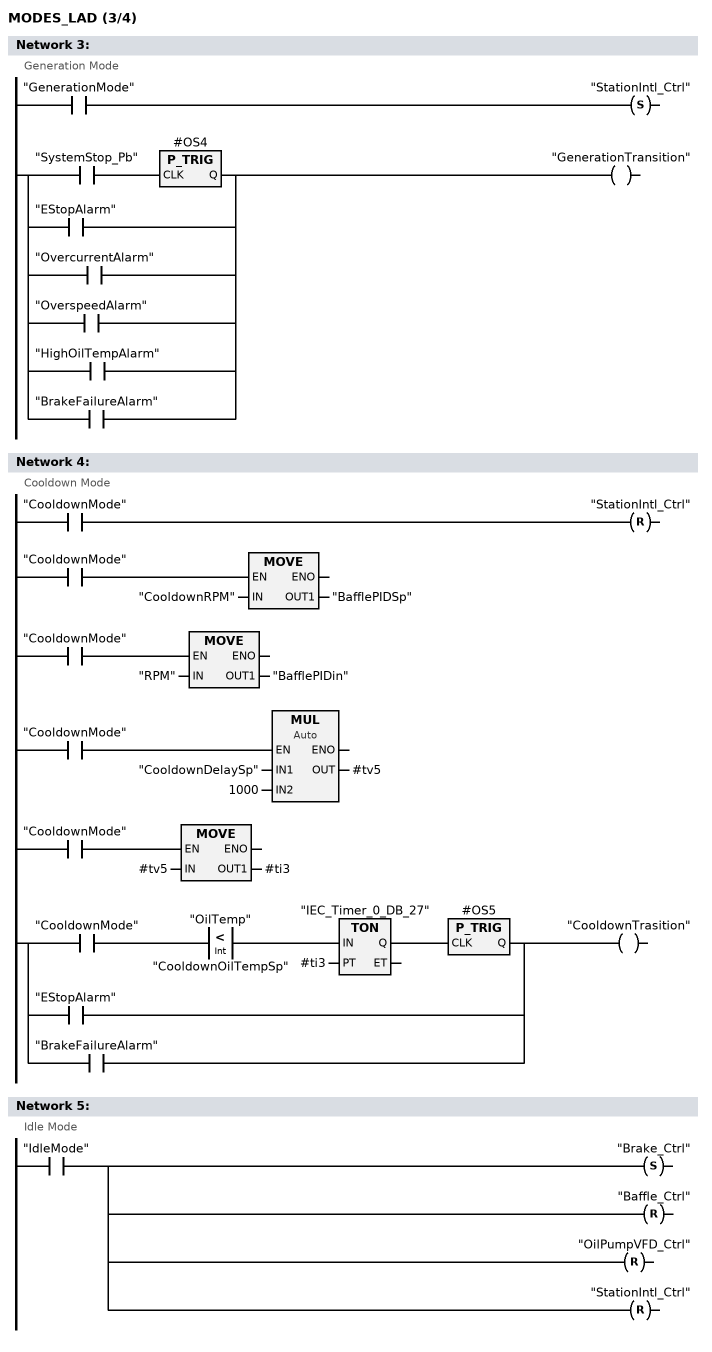
   RUNG wire#powerrail
      Contact( "GenerationMode" )
      S_Coil( "StationIntl_Ctrl" )
   END_RUNG
   RUNG wire#powerrail
      Contact( "SystemStop_Pb" )
      P_Trig( #OS4 )
      wire#w1
      Coil( "GenerationTransition" )
   END_RUNG
   RUNG wire#powerrail
      Contact( "EStopAlarm" )
   END_RUNG wire#w1
   RUNG wire#powerrail
      Contact( "OvercurrentAlarm" )
   END_RUNG wire#w1
   RUNG wire#powerrail
      Contact( "OverspeedAlarm" )
   END_RUNG wire#w1
   RUNG wire#powerrail
      Contact( "HighOilTempAlarm" )
   END_RUNG wire#w1
   RUNG wire#powerrail
      Contact( "BrakeFailureAlarm" )
   END_RUNG wire#w1
   // the same network as SCL:
   IF "GenerationMode" THEN "StationIntl_Ctrl" := TRUE; END_IF;
   #_w1 := "SystemStop_Pb" AND NOT #OS4;   // rising edge
   #OS4 := "SystemStop_Pb";
   "GenerationTransition" := #_w1 OR "EStopAlarm" OR "OvercurrentAlarm" OR "OverspeedAlarm" OR "HighOilTempAlarm" OR "BrakeFailureAlarm";
END_REGION

REGION Network 4
   // Cooldown Mode
   IF "CooldownMode" THEN
       "StationIntl_Ctrl" := FALSE;
       "BafflePIDSp" := "CooldownRPM";
       "BafflePIDin" := "RPM";
       #tv5 := "CooldownDelaySp" * 1000;
       #ti3 := #tv5;
   END_IF;
   "IEC_Timer_0_DB_27".TON(IN := "CooldownMode" AND ("OilTemp" < "CooldownOilTempSp"), PT := #ti3);
   #_w1 := "IEC_Timer_0_DB_27".Q AND NOT #OS5;   // rising edge
   #OS5 := "IEC_Timer_0_DB_27".Q;
   "CooldownTrasition" := #_w1 OR "EStopAlarm" OR "BrakeFailureAlarm";
END_REGION

REGION Network 5
   // Idle Mode
   RUNG wire#powerrail
      Contact( "IdleMode" )
      wire#w1
      S_Coil( "Brake_Ctrl" )
   END_RUNG
   RUNG wire#w1
      R_Coil( "Baffle_Ctrl" )
   END_RUNG
   RUNG wire#w1
      R_Coil( "OilPumpVFD_Ctrl" )
   END_RUNG
   RUNG wire#w1
      R_Coil( "StationIntl_Ctrl" )
   END_RUNG
   // the same network as SCL:
   IF "IdleMode" THEN
       "Brake_Ctrl" := TRUE;
       "Baffle_Ctrl" := FALSE;
       "OilPumpVFD_Ctrl" := FALSE;
       "StationIntl_Ctrl" := FALSE;
   END_IF;
END_REGION

REGION Network 6
   // Fault Mode
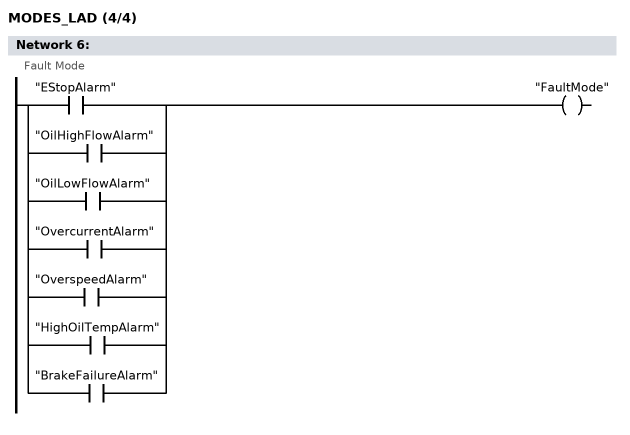
   RUNG wire#powerrail
      Contact( "EStopAlarm" )
      wire#w1
      Coil( "FaultMode" )
   END_RUNG
   RUNG wire#powerrail
      Contact( "OilHighFlowAlarm" )
   END_RUNG wire#w1
   RUNG wire#powerrail
      Contact( "OilLowFlowAlarm" )
   END_RUNG wire#w1
   RUNG wire#powerrail
      Contact( "OvercurrentAlarm" )
   END_RUNG wire#w1
   RUNG wire#powerrail
      Contact( "OverspeedAlarm" )
   END_RUNG wire#w1
   RUNG wire#powerrail
      Contact( "HighOilTempAlarm" )
   END_RUNG wire#w1
   RUNG wire#powerrail
      Contact( "BrakeFailureAlarm" )
   END_RUNG wire#w1
   // the same network as SCL:
   "FaultMode" := "EStopAlarm" OR "OilHighFlowAlarm" OR "OilLowFlowAlarm" OR "OvercurrentAlarm" OR "OverspeedAlarm" OR "HighOilTempAlarm" OR "BrakeFailureAlarm";
END_REGION
END_FUNCTION_BLOCK

FUNCTION_BLOCK "MODES_FBD"   // FB15, FBD
{ S7_Optimized_Access := 'TRUE' }
VERSION : 0.1
   VAR
      OS1 : Bool;
      OS2 : Bool;
      OS3 : Bool;
      OS4 : Bool;
      OS5 : Bool;
   END_VAR
   VAR_TEMP
      ti1 : Time;
      tv1 : Int;
      tv2 : Int;
      ti3 : Time;
      ti2 : Time;
   END_VAR
   VAR_TEMP   // added for the SCL form of the ladder/FBD networks
      _w1 : Bool;
      _w2 : Bool;
      _w3 : Bool;
   END_VAR
BEGIN

REGION Network 1
   // Warmup Mode
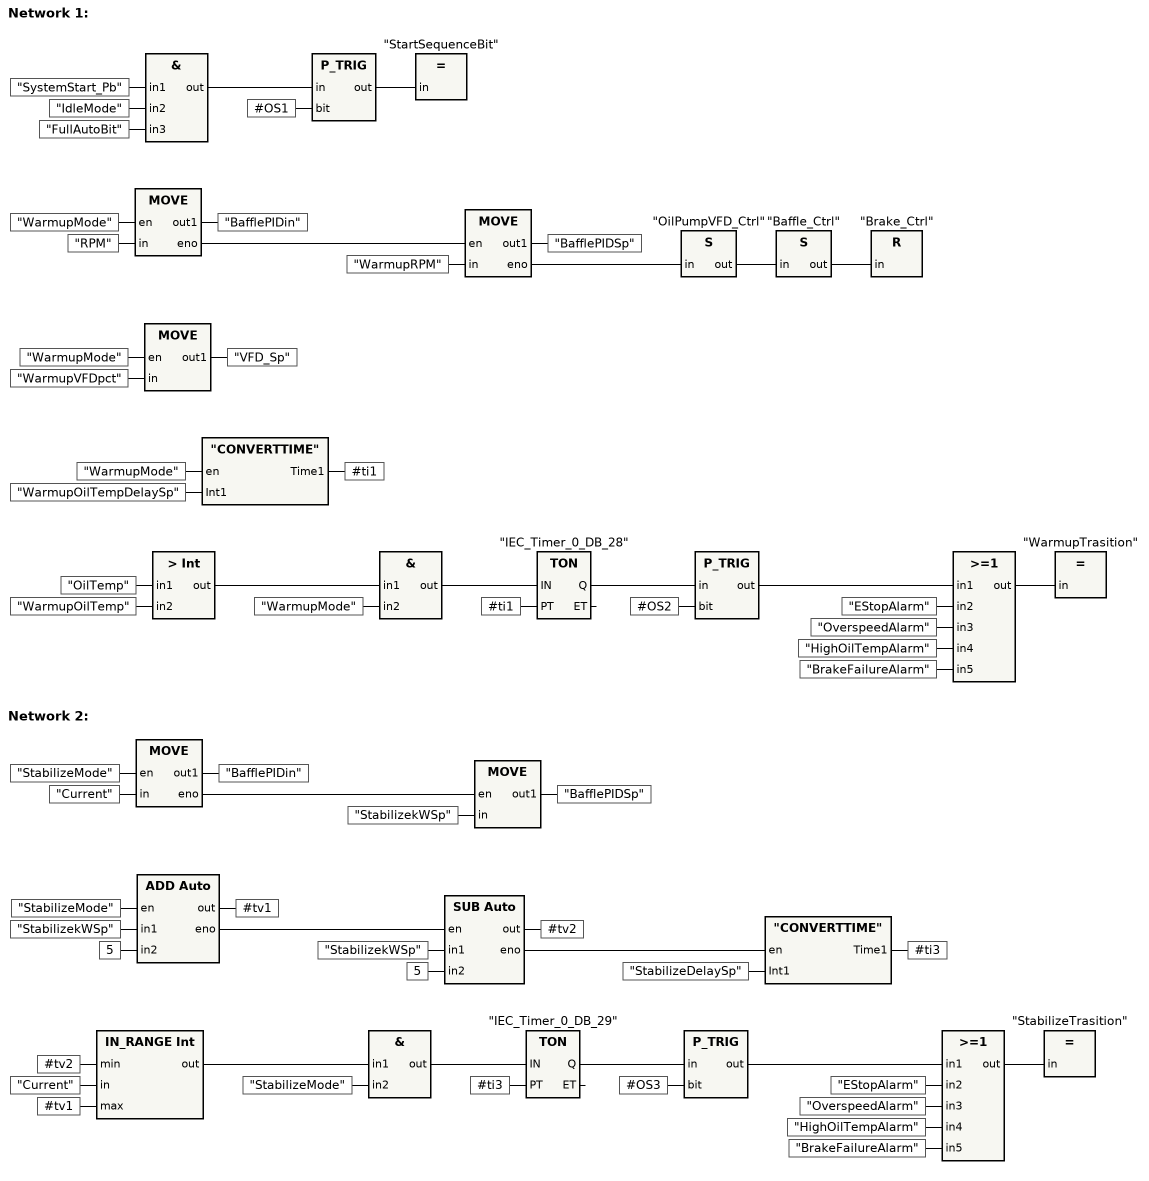
   #_w1 := "SystemStart_Pb" AND "IdleMode" AND "FullAutoBit";
   #_w2 := #_w1 AND NOT #OS1;   // rising edge
   #OS1 := #_w1;
   "StartSequenceBit" := #_w2;
   IF "WarmupMode" THEN
       "BafflePIDin" := "RPM";
       "BafflePIDSp" := "WarmupRPM";
       "OilPumpVFD_Ctrl" := TRUE;
       "Baffle_Ctrl" := TRUE;
       "Brake_Ctrl" := FALSE;
       "VFD_Sp" := "WarmupVFDpct";
       "CONVERTTIME"(Int1 := "WarmupOilTempDelaySp", Time1 => #ti1);
   END_IF;
   "IEC_Timer_0_DB_28".TON(IN := ("OilTemp" > "WarmupOilTemp") AND "WarmupMode", PT := #ti1);
   #_w3 := "IEC_Timer_0_DB_28".Q AND NOT #OS2;   // rising edge
   #OS2 := "IEC_Timer_0_DB_28".Q;
   "WarmupTrasition" := #_w3 OR "EStopAlarm" OR "OverspeedAlarm" OR "HighOilTempAlarm" OR "BrakeFailureAlarm";
END_REGION

REGION Network 2
   // Stabilize Mode
   IF "StabilizeMode" THEN
       "BafflePIDin" := "Current";
       "BafflePIDSp" := "StabilizekWSp";
       #tv1 := "StabilizekWSp" + 5;
       #tv2 := "StabilizekWSp" - 5;
       "CONVERTTIME"(Int1 := "StabilizeDelaySp", Time1 => #ti3);
   END_IF;
   "IEC_Timer_0_DB_29".TON(IN := (#tv2 <= "Current") AND ("Current" <= #tv1) AND "StabilizeMode", PT := #ti3);
   #_w1 := "IEC_Timer_0_DB_29".Q AND NOT #OS3;   // rising edge
   #OS3 := "IEC_Timer_0_DB_29".Q;
   "StabilizeTrasition" := #_w1 OR "EStopAlarm" OR "OverspeedAlarm" OR "HighOilTempAlarm" OR "BrakeFailureAlarm";
END_REGION

REGION Network 3
   // Generation Mode
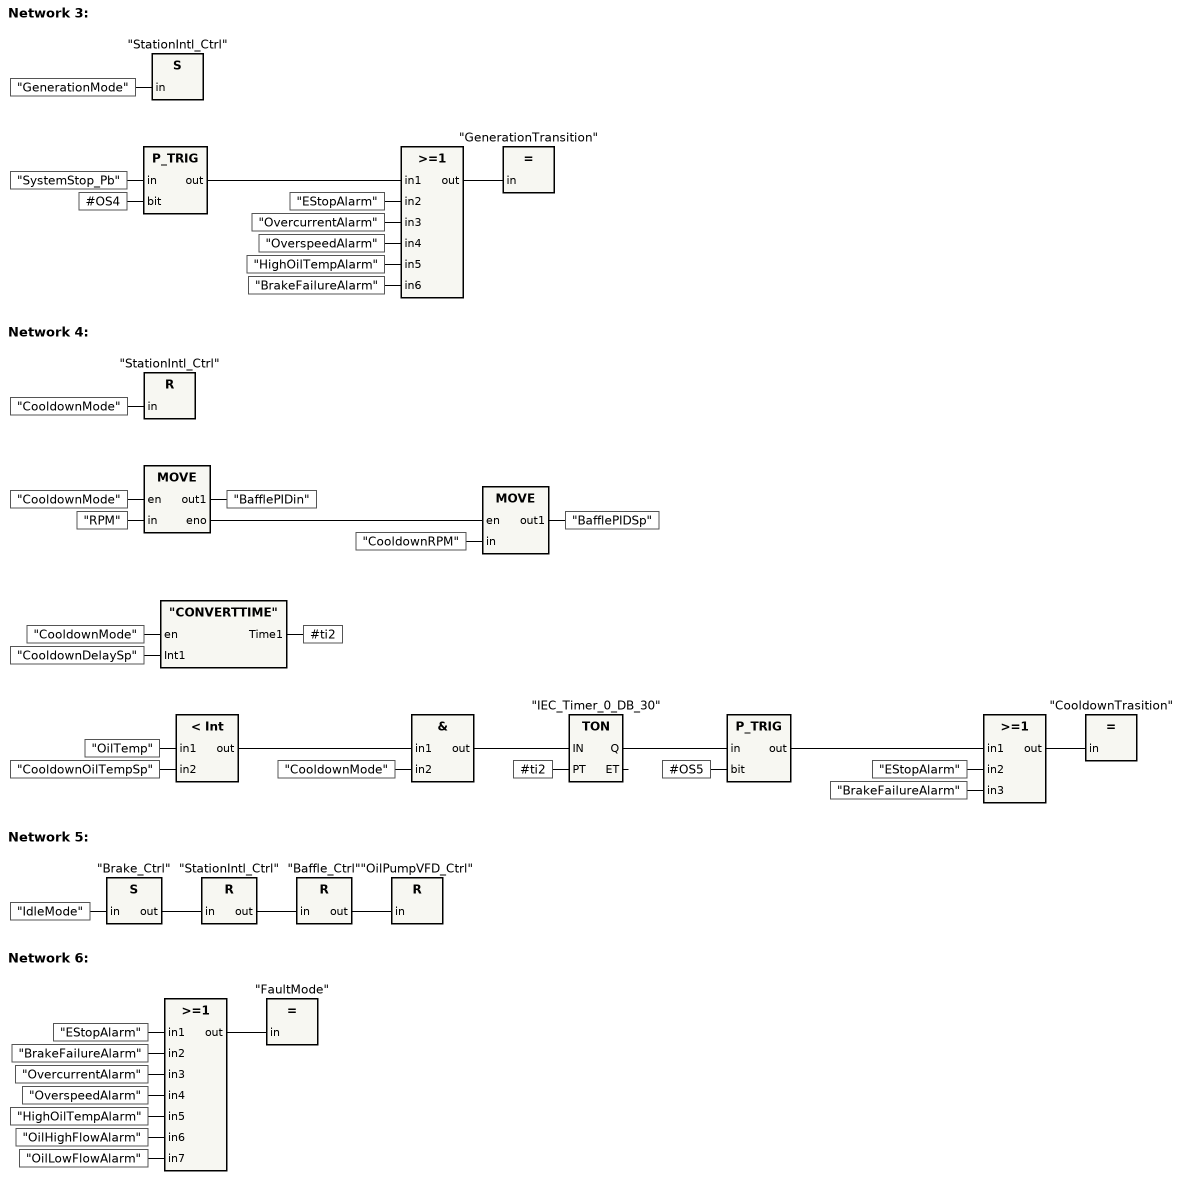
   IF "GenerationMode" THEN "StationIntl_Ctrl" := TRUE; END_IF;
   #_w1 := "SystemStop_Pb" AND NOT #OS4;   // rising edge
   #OS4 := "SystemStop_Pb";
   "GenerationTransition" := #_w1 OR "EStopAlarm" OR "OvercurrentAlarm" OR "OverspeedAlarm" OR "HighOilTempAlarm" OR "BrakeFailureAlarm";
END_REGION

REGION Network 4
   // Cooldown Mode
   IF "CooldownMode" THEN
       "StationIntl_Ctrl" := FALSE;
       "BafflePIDin" := "RPM";
       "BafflePIDSp" := "CooldownRPM";
       "CONVERTTIME"(Int1 := "CooldownDelaySp", Time1 => #ti2);
   END_IF;
   "IEC_Timer_0_DB_30".TON(IN := ("OilTemp" < "CooldownOilTempSp") AND "CooldownMode", PT := #ti2);
   #_w1 := "IEC_Timer_0_DB_30".Q AND NOT #OS5;   // rising edge
   #OS5 := "IEC_Timer_0_DB_30".Q;
   "CooldownTrasition" := #_w1 OR "EStopAlarm" OR "BrakeFailureAlarm";
END_REGION

REGION Network 5
   // Idle Mode
   IF "IdleMode" THEN
       "Brake_Ctrl" := TRUE;
       "StationIntl_Ctrl" := FALSE;
       "Baffle_Ctrl" := FALSE;
       "OilPumpVFD_Ctrl" := FALSE;
   END_IF;
END_REGION

REGION Network 6
   // Fault Mode
   "FaultMode" := "EStopAlarm" OR "BrakeFailureAlarm" OR "OvercurrentAlarm" OR "OverspeedAlarm" OR "HighOilTempAlarm" OR "OilHighFlowAlarm" OR "OilLowFlowAlarm";
END_REGION
END_FUNCTION_BLOCK

FUNCTION_BLOCK "MODES_SCL"   // FB16, SCL
{ S7_Optimized_Access := 'TRUE' }
VERSION : 0.1
   VAR_TEMP
      ti1 : Time;
      ti2 : Time;
      tv1 : Int;
      tv2 : Int;
      ti3 : Time;
      warmupdelaytrigger : Bool;
      stabilizedelaytrigger : Bool;
      ti4 : Time;
      ti5 : Time;
      cooldowndelaytrigger : Bool;
      ti6 : Time;
   END_VAR
BEGIN
   //EStop Handling
   IF "EStopAlarm" OR "BrakeFailureAlarm" THEN
       "WarmupTrasition" := 1;
       "StabilizeTrasition" := 1;
       "GenerationTransition" := 1;
       "CooldownTrasition" := 1;
   ELSE
       "WarmupTrasition" := 0;
       "StabilizeTrasition" := 0;
       "GenerationTransition" := 0;
       "CooldownTrasition" := 0;

       //Warmup Mode
       IF "SystemStart_Pb" AND "IdleMode" AND "FullAutoBit" THEN
           "StartSequenceBit" := 1;
       ELSE
           "StartSequenceBit" := 0;
       END_IF;


       IF "WarmupMode" THEN
           "Brake_Ctrl" := 0;
           "Baffle_Ctrl" := 1;
           "OilPumpVFD_Ctrl" := 1;
           "BafflePIDin" := "RPM";
           "BafflePIDSp" := "WarmupRPM";
           "VFD_Sp" := "WarmupVFDpct";
           IF "OilTemp" > "WarmupOilTemp" THEN
               "CONVERTTIME"(Int1 := "WarmupOilTempDelaySp",
                             Time1 => #ti1);
               "IEC_Timer_0_DB_31".TON(IN := TRUE,
                                       PT := #ti1,
                                       Q => #warmupdelaytrigger,
                                       ET => #ti2);
           ELSE
               RESET_TIMER("IEC_Timer_0_DB_31");
           END_IF;
           IF #warmupdelaytrigger THEN
               RESET_TIMER("IEC_Timer_0_DB_31");
               "WarmupTrasition" := 1;
           END_IF;
       ELSE
           "WarmupTrasition" := 0;
       END_IF;

       IF "OverspeedAlarm" OR "HighOilTempAlarm" THEN
           "WarmupTrasition" := 1;
       END_IF;

       //Stabilize Mode
       IF "StabilizeMode" THEN
           "BafflePIDin" := "Current";
           "BafflePIDSp" := "StabilizekWSp";
           #tv1 := "StabilizekWSp" - 5;
           #tv2 := "StabilizekWSp" + 5;
           IF "Current" < #tv2 AND "Current" > #tv1 THEN
               "CONVERTTIME"(Int1 := "StabilizeDelaySp",
                             Time1 => #ti3);
               "IEC_Timer_0_DB_32".TON(IN := TRUE,
                                       PT := #ti3,
                                       Q => #stabilizedelaytrigger,
                                       ET => #ti4);
           ELSE
               RESET_TIMER("IEC_Timer_0_DB_32");
           END_IF;
           IF #stabilizedelaytrigger THEN
               RESET_TIMER("IEC_Timer_0_DB_31");
               "StabilizeTrasition" := 1;
           END_IF;
       ELSE
           "StabilizeTrasition" := 0;
       END_IF;

       IF "OverspeedAlarm" OR "HighOilTempAlarm" THEN
           "StabilizeTrasition" := 1;
       END_IF;


       //Generation Mode
       IF "GenerationMode" THEN
           "StationIntl_Ctrl" := 1;
           IF "SystemStop_Pb" THEN
               "GenerationTransition" := 1;
           END_IF;
       ELSE
           "GenerationTransition" := 0;
       END_IF;

       IF "OvercurrentAlarm" OR "OverspeedAlarm" OR "HighOilTempAlarm" THEN
           "GenerationTransition" := 1;
       END_IF;


       //Cooldown Mode
       IF "CooldownMode" THEN
           "StationIntl_Ctrl" := 0;
           "BafflePIDin" := "RPM";
           "BafflePIDSp" := "CooldownRPMSp";
           IF "OilTemp" < "CooldownOilTempSp" THEN
               "CONVERTTIME"(Int1 := "CooldownDelaySp",
                             Time1 => #ti5);
               "IEC_Timer_0_DB_33".TON(IN := TRUE,
                                       PT := #ti5,
                                       Q => #cooldowndelaytrigger,
                                       ET => #ti6);
           ELSE
               RESET_TIMER("IEC_Timer_0_DB_33");
           END_IF;
           IF #cooldowndelaytrigger THEN
               RESET_TIMER("IEC_Timer_0_DB_33");
               "CooldownTrasition" := 1;
           END_IF;
       ELSE
           "CooldownTrasition" := 0;
       END_IF;


       //Fault Mode
       IF "EStopAlarm" OR "BrakeFailureAlarm" OR "OvercurrentAlarm" OR "OverspeedAlarm" OR "HighOilTempAlarm" OR "OilHighFlowAlarm" OR "OilLowFlowAlarm" THEN
           "FaultMode" := 1;
       ELSE
           "FaultMode" := 0;
       END_IF;

   END_IF;

   //Idle Mode
   IF "IdleMode" THEN
       "Brake_Ctrl" := 1;
       "OilPumpVFD_Ctrl" := 0;
       "Baffle_Ctrl" := 0;
       "StationIntl_Ctrl" := 0;
   END_IF;
END_FUNCTION_BLOCK

FUNCTION_BLOCK "MODES_STL"   // FB17, STL
{ S7_Optimized_Access := 'TRUE' }
VERSION : 0.1
   VAR
      OS1 : Bool;
      OS2 : Bool;
   END_VAR
   VAR_TEMP
      ti1 : Time;
      warmupdelaytrigger : Bool;
      ti2 : Time;
      tv1 : Int;
      tv2 : Int;
      tb1 : Bool;
      ti3 : Time;
      stabilizedelaytrigger : Bool;
      ti4 : Time;
      ti5 : Time;
      ti6 : Time;
      cooldowndelaytrigger : Bool;
   END_VAR
BEGIN

REGION Network 1
   //EStop Handling
   EStop:A     "EStopAlarm";
         O     "BrakeFailureAlarm";
         JC    EStopTransitions;
         JU    ResetTransitions;

   EStopTransitions:SET;
         S     "WarmupTrasition";
         S     "StabilizeTrasition";
         S     "GenerationTransition";
         S     "CooldownTrasition";
         JU    JumpToMode;

   ResetTransitions:CLR;
         NOT;
         R     "WarmupTrasition";
         R     "StabilizeTrasition";
         R     "GenerationTransition";
         R     "CooldownTrasition";
         JU    JumpToMode;

   JumpToMode:A     "WarmupMode";
         JC    StartWarmup;
         CLR;
         A     "StabilizeMode";
         JC    StabilizeMode;
         CLR;
         A     "GenerationMode";
         JC    GenerationMode;
         CLR;
         A     "CooldownMode";
         JC    CooldownMode;
         CLR;
         A     "IdleMode";
         JC    IdleMode;
         JU    EndOfLine;

   //Warmup Mode
   StartWarmup:SET;
         R     "WarmupTrasition";
         R     "StabilizeTrasition";
         R     "GenerationTransition";
         R     "CooldownTrasition";
         R     "StartSequenceBit";
         CLR;
         A     "WarmupMode";
         JC    WarmupMode;
         CLR;
         A     "StabilizeMode";
         JC    StabilizeMode;
         CLR;
         A     "GenerationMode";
         JC    GenerationMode;
         CLR;
         A     "CooldownMode";
         JC    CooldownMode;
         CLR;
         A     "IdleMode";
         JC    IdleMode;
         JU    EndOfLine;

   WarmupMode:SET;
         NOT;
         R     "Brake_Ctrl";
         L     "WarmupRPM";
         T     "BafflePIDSp";
         L     "RPM";
         T     "BafflePIDin";

         SET;
         S     "OilPumpVFD_Ctrl";
         S     "Baffle_Ctrl";
         L     "WarmupVFDpct";
         T     "VFD_Sp";

         L     "OilTemp";
         L     "WarmupOilTemp";
         >I;
         JC    WarmupTime;
         CALL  RESET_TIMER
         ( "TIMER" := "IEC_Timer_0_DB_34"
         );
         JU    StabilizeMode;

   WarmupTime:CALL  "CONVERTTIME"
         ( Int1  := "WarmupOilTempDelaySp",
           Time1 := #ti1
         );
         CALL  TON, "IEC_Timer_0_DB_34"
         ( IN := TRUE,
           PT := #ti1,
           Q  := #warmupdelaytrigger,
           ET := #ti2
         );
         A     #warmupdelaytrigger;
         JC    WarmupExit;
         CLR;
         A     "OverspeedAlarm";
         O     "HighOilTempAlarm";
         JC    WarmupExit;
         JU    StabilizeMode;

   WarmupExit:S     "WarmupTrasition";
         CALL  RESET_TIMER
         ( "TIMER" := "IEC_Timer_0_DB_34"
         );
         JU    StabilizeMode;

   //Stabilize Mode
   StabilizeMode:SET;
         NOT;
         R     "WarmupTrasition";
         L     "StabilizekWSp";
         T     "BafflePIDSp";
         L     "Current";
         T     "BafflePIDin";
         L     "StabilizekWSp";
         L     5;
         +I;
         T     #tv1;
         L     "StabilizekWSp";
         L     5;
         -I;
         T     #tv2;
         L     "Current";
         L     #tv1;
         <I;
         S     #tb1;
         L     "Current";
         L     #tv2;
         >I;
         A     #tb1;
         JC    StabilizeTime;
         CALL  RESET_TIMER
         ( "TIMER" := "IEC_Timer_0_DB_35"
         );
         JU    GenerationMode;

   StabilizeTime:CALL  "CONVERTTIME"
         ( Int1  := "StabilizeDelaySp",
           Time1 := #ti3
         );
         CALL  TON , "IEC_Timer_0_DB_35"
         ( IN := TRUE,
           PT := #ti3,
           Q  := #stabilizedelaytrigger,
           ET := #ti4
         );
         A     #stabilizedelaytrigger;
         JC    StabilizeExit;
         CLR;
         A     "OverspeedAlarm";
         O     "HighOilTempAlarm";
         JC    StabilizeExit;
         JU    GenerationMode;

   StabilizeExit:S     "StabilizeTrasition";
         CALL  RESET_TIMER
         ( "TIMER" := "IEC_Timer_0_DB_35"
         );
         JU    GenerationMode;

   //Generation Mode
   GenerationMode:SET;
         NOT;
         R     "StabilizeTrasition";
         SET;
         S     "StationIntl_Ctrl";
         A     "SystemStop_Pb";
         JC    GenerationExit;
         CLR;
         A     "OvercurrentAlarm";
         JC    GenerationExit;
         CLR;
         A     "OverspeedAlarm";
         O     "HighOilTempAlarm";
         JC    GenerationExit;
         JU    CooldownMode;

   GenerationExit:S     "GenerationTransition";
         JU    CooldownMode;

   // Cooldown Mode
   CooldownMode:SET;
         NOT;
         R     "GenerationTransition";
         R     "StationIntl_Ctrl";
         L     "CooldownRPM";
         T     "BafflePIDSp";
         L     "RPM";
         T     "BafflePIDin";
         L     "OilTemp";
         L     "CooldownOilTempSp";
         <I;
         JC    CooldownTime;
         CALL  RESET_TIMER
         ( "TIMER" := "IEC_Timer_0_DB_36"
         );
         JU    IdleMode;

   CooldownTime:CALL  "CONVERTTIME"
         ( Int1  := "CooldownDelaySp",
           Time1 := #ti5
         );
         CALL  TON , "IEC_Timer_0_DB_36"
         ( IN := TRUE,
           PT := #ti5,
           Q  := #cooldowndelaytrigger,
           ET := #ti6
         );
         A     #cooldowndelaytrigger;
         JC    CooldownExit;
         JU    IdleMode;

   CooldownExit:S     "CooldownTrasition";
         CALL  RESET_TIMER
         ( "TIMER" := "IEC_Timer_0_DB_36"
         );
         JU    IdleMode;


   //Idle Mode
   IdleMode:SET;
         NOT;
         R     "CooldownTrasition";
         R     "StationIntl_Ctrl";
         S     "Brake_Ctrl";
         R     "Baffle_Ctrl";
         R     "OilPumpVFD_Ctrl";
         CLR;
         A     "SystemStart_Pb";
         A     "IdleMode";
         A     "FullAutoBit";
         FP    #OS1;
         S     "StartSequenceBit";
         JU    EndOfLine;

   //Fault Mode
   EndOfLine:A     "EStopAlarm";
         O     "BrakeFailureAlarm";
         O     "OvercurrentAlarm";
         O     "OverspeedAlarm";
         O     "HighOilTempAlarm";
         O     "OilHighFlowAlarm";
         O     "OilLowFlowAlarm";
         =     "FaultMode";
END_REGION
END_FUNCTION_BLOCK

FUNCTION_BLOCK "SEQUENCE"   // FB18, GRAPH_PLUS
{ S7_Optimized_Access := 'TRUE' }
VERSION : 0.1
   VAR_INPUT
      OFF_SQ : Bool := false;   // Turn sequence off
      INIT_SQ : Bool := false;   // Set sequence to initial state
      ACK_EF : Bool := false;   // Acknowledge all errors and faults
      S_PREV : Bool := false;   // Output previous step in parameter S_NO
      S_NEXT : Bool := false;   // Indicate next step in parameter S_NO
      SW_AUTO : Bool := false;   // Automatic mode
      SW_TAP : Bool := false;   // Semiautomatic/switch with transition
      SW_TOP : Bool := false;   // Semiautomatic/ignore transition
      SW_MAN : Bool := false;   // Manual mode
      S_SEL : Int := 0;   // Select step to be output to S_NO
      S_ON : Bool := false;   // Activate step indicated in S_NO
      S_OFF : Bool := false;   // Deactivate step indicated S_NO
      T_PUSH : Bool := false;   // Enable transition to switch in semi automatic mode
   END_VAR
   VAR_OUTPUT
      S_NO : Int := 0;   // Step number
      S_MORE : Bool := false;   // More steps are available and can be shown in S_NO
      S_ACTIVE : Bool := false;   // Step indicated in S_NO is active
      ERR_FLT : Bool := false;   // Interlock or supervision group error
      AUTO_ON : Bool := false;   // Automatic mode is active
      TAP_ON : Bool := false;   // Semiautomatic mode/step with transition enabled
      TOP_ON : Bool := false;   // Semiautomatic mode/ignore transition enabled
      MAN_ON : Bool := false;   // Manual mode is active
   END_VAR
   VAR
      HMI_INFO : Array[0..8] of UInt;
      IF_PAR : G7_IfParPlus_V2;
      RT_DATA : G7_RTDataPlus_V2;   // Internal data area
      Trans1 : G7_TransitionPlus_V2;   // Transition structure
      Trans2 : G7_TransitionPlus_V2;   // Transition structure
      Trans3 : G7_TransitionPlus_V2;   // Transition structure
      Trans4 : G7_TransitionPlus_V2;   // Transition structure
      Trans5 : G7_TransitionPlus_V2;   // Transition structure
      Idle : G7_StepPlus_V2;   // Step structure
      Warmup : G7_StepPlus_V2;   // Step structure
      Stabilize : G7_StepPlus_V2;   // Step structure
      Generation : G7_StepPlus_V2;   // Step structure
      Cooldown : G7_StepPlus_V2;   // Step structure
      SINI : Array[0..1] of USInt;
      LSTT : Array[0..4] of USInt;
      ATAJ : Array[0..4] of USInt;
      ATAB : Array[0..4] of USInt;
      PSTT : Array[0..4] of USInt;
      NSTT : Array[0..4] of USInt;
      ASSJ : Array[0..4] of USInt;
      ASSB : Array[0..4] of USInt;
      PTTS : Array[0..4] of USInt;
      NTTS : Array[0..4] of USInt;
      SW_SQTS : Array[0..4] of USInt;
      SWITCH : Array[0..0] of USInt;
      TVX : Array[0..1] of USInt;
      TTX : Array[0..1] of USInt;
      TSX : Array[0..1] of USInt;
      S00X : Array[0..1] of USInt;
      SOFFX : Array[0..1] of USInt;
      SONX : Array[0..1] of USInt;
      SAX : Array[0..1] of USInt;
      SERRX : Array[0..5] of USInt;
      SMX : Array[0..5] of USInt;
      S0X : Array[0..5] of USInt;
      S1X : Array[0..5] of USInt;
      IL_ALARM_INST : Program_Alarm;
      SUP_ALARM_INST : Program_Alarm;
      STEP_TIME_ALARM_INST : Program_Alarm;
      IEC_TIMER_INST : IEC_TIMER;
      TRANSACTION_FLAG : Bool := false;
   END_VAR
   // SINI[0] := 2;
   // SINI[1] := 1;
   // LSTT[0] := 255;
   // LSTT[1] := 255;
   // LSTT[2] := 255;
   // LSTT[4] := 255;
   // ATAJ[1] := 1;
   // ATAJ[2] := 2;
   // ATAJ[3] := 3;
   // ATAJ[4] := 4;
   // ATAB[1] := 1;
   // ATAB[2] := 2;
   // ATAB[3] := 3;
   // ATAB[4] := 4;
   // PSTT[0] := 1;
   // PSTT[1] := 2;
   // PSTT[2] := 3;
   // PSTT[3] := 4;
   // NSTT[0] := 2;
   // NSTT[1] := 3;
   // NSTT[2] := 4;
   // NSTT[4] := 1;
   // ASSJ[1] := 1;
   // ASSJ[2] := 2;
   // ASSJ[3] := 3;
   // ASSJ[4] := 4;
   // ASSB[1] := 1;
   // ASSB[2] := 2;
   // ASSB[3] := 3;
   // ASSB[4] := 4;
   // PTTS[0] := 255;
   // PTTS[1] := 4;
   // PTTS[3] := 1;
   // PTTS[4] := 2;
   // NTTS[0] := 4;
   // NTTS[2] := 1;
   // NTTS[3] := 2;
   // NTTS[4] := 3;
   // TVX[0] := 16#1;
   // TTX[0] := 16#1;
   // TSX[0] := 16#1;
   // S00X[0] := 16#1;
   // SOFFX[0] := 16#1;
   // SONX[0] := 16#1;
   // SAX[0] := 16#1;
   // SERRX[0] := 16#1;
   // SMX[0] := 16#1;
   // S0X[0] := 16#1;
   // S1X[0] := 16#1;
BEGIN
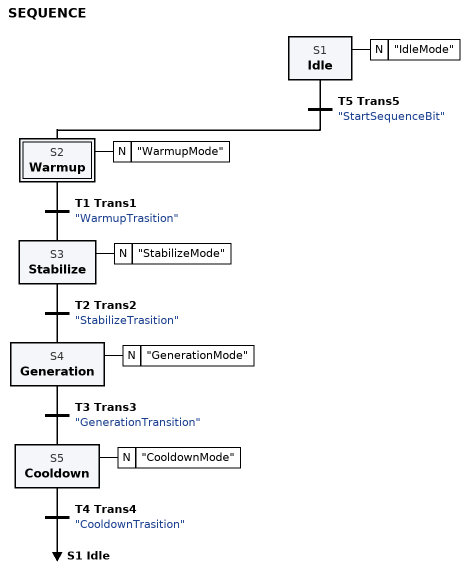
   // sequencer 1
   STEP Idle:   // S1, max time T#10S, warning time T#7S
              N    "IdleMode"
   END_STEP
   TRANSITION Trans5 FROM Idle TO Warmup   // T5
      := "StartSequenceBit";
   END_TRANSITION
   INITIAL_STEP Warmup:   // S2, max time T#10S, warning time T#7S
              N    "WarmupMode"
   END_STEP
   TRANSITION Trans1 FROM Warmup TO Stabilize   // T1
      := "WarmupTrasition";
   END_TRANSITION
   STEP Stabilize:   // S3, max time T#10S, warning time T#7S
              N    "StabilizeMode"
   END_STEP
   TRANSITION Trans2 FROM Stabilize TO Generation   // T2
      := "StabilizeTrasition";
   END_TRANSITION
   STEP Generation:   // S4, max time T#10S, warning time T#7S
              N    "GenerationMode"
   END_STEP
   TRANSITION Trans3 FROM Generation TO Cooldown   // T3
      := "GenerationTransition";
   END_TRANSITION
   STEP Cooldown:   // S5, max time T#10S, warning time T#7S
              N    "CooldownMode"
   END_STEP
   TRANSITION Trans4 FROM Cooldown TO Idle   // T4, jump
      := "CooldownTrasition";
   END_TRANSITION
END_FUNCTION_BLOCK

FUNCTION_BLOCK "HOURMETER_LAD"   // FB19, LAD
{ S7_Optimized_Access := 'TRUE' }
VERSION : 0.1
   VAR
      accum_elapsed : Time;
      OS1 : Bool;
      MinuteTimedDown : Bool;
      HourCountedDown : Bool;
      OS2 : Bool;
      OS3 : Bool;
      DayCountedDown : Bool;
      resettime : Time;
      OS4 : Bool;
      resetrto : Bool;
      minutecounterreset : Bool;
      hourcounterreset : Bool;
   END_VAR
   VAR_TEMP
      resethourmetertrigger : Bool;
   END_VAR
   VAR_TEMP   // added for the SCL form of the ladder/FBD networks
      _w1 : Bool;
      _w2 : Bool;
      _w3 : Bool;
   END_VAR
BEGIN

REGION Network 1
